REGION Network 56: Step[1130] : Gripper Forward
   RUNG wire#powerrail
      { S7_Templates := "SrcType := DInt" } EQ_Contact(in1 := "Unit1.Em7.ControlNodes".sepaGripper.sequence.status.currentStep, in2 := #JOB_11_STEP_30)
      Contact( "Unit1.Em7.ControlNodes".sepaGripper.sequence.status.seqActive )
      wire#w1
      Coil( "Unit1.Em7.ControlNodes".sepaGripper."step".action1[1130] )
   END_RUNG
   RUNG wire#w1
      Contact( "Unit1.Em7.ControlNodes".cmStackGripperFwdBwd.monitoring.inWorkPos )
      Coil( "Unit1.Em7.ControlNodes".sepaGripper."step".transition1[1130] )
   END_RUNG
   RUNG wire#w1
      Contact( "Unit1.Em7.ControlNodes".sepaGripper."step".transition1[1130] )
      Move(in := #JOB_11_STEP_40, out1 => "Unit1.Em7.ControlNodes".sepaGripper.sequence.status.nextStep)
   END_RUNG
   // the same network as SCL:
   "Unit1.Em7.ControlNodes".sepaGripper."step".action1[1130] := ("Unit1.Em7.ControlNodes".sepaGripper.sequence.status.currentStep = #JOB_11_STEP_30) AND "Unit1.Em7.ControlNodes".sepaGripper.sequence.status.seqActive;
   "Unit1.Em7.ControlNodes".sepaGripper."step".transition1[1130] := ("Unit1.Em7.ControlNodes".sepaGripper.sequence.status.currentStep = #JOB_11_STEP_30) AND "Unit1.Em7.ControlNodes".sepaGripper.sequence.status.seqActive AND "Unit1.Em7.ControlNodes".cmStackGripperFwdBwd.monitoring.inWorkPos;
   IF ("Unit1.Em7.ControlNodes".sepaGripper.sequence.status.currentStep = #JOB_11_STEP_30) AND "Unit1.Em7.ControlNodes".sepaGripper.sequence.status.seqActive AND "Unit1.Em7.ControlNodes".sepaGripper."step".transition1[1130] THEN
       "Unit1.Em7.ControlNodes".sepaGripper.sequence.status.nextStep := #JOB_11_STEP_40;
   END_IF;
END_REGION

REGION Network 57: Step[1140] : Gripper X-Axis Grip Pos
   RUNG wire#powerrail
      { S7_Templates := "SrcType := DInt" } EQ_Contact(in1 := "Unit1.Em7.ControlNodes".sepaGripper.sequence.status.currentStep, in2 := #JOB_11_STEP_40)
      Contact( "Unit1.Em7.ControlNodes".sepaGripper.sequence.status.seqActive )
      wire#w1
      Coil( "Unit1.Em7.ControlNodes".sepaGripper."step".action1[1140] )
   END_RUNG
   RUNG wire#w1
      Contact( "Unit1.Em7.ControlNodes".cm.softCam.sepaGripperAxisX.pickUpPOs.inPos )
      Coil( "Unit1.Em7.ControlNodes".sepaGripper."step".transition1[1140] )
   END_RUNG
   RUNG wire#w1
      Contact( "Unit1.Em7.ControlNodes".sepaGripper."step".transition1[1140] )
      Move(in := #JOB_11_STEP_90, out1 => "Unit1.Em7.ControlNodes".sepaGripper.sequence.status.nextStep)
   END_RUNG
   // the same network as SCL:
   "Unit1.Em7.ControlNodes".sepaGripper."step".action1[1140] := ("Unit1.Em7.ControlNodes".sepaGripper.sequence.status.currentStep = #JOB_11_STEP_40) AND "Unit1.Em7.ControlNodes".sepaGripper.sequence.status.seqActive;
   "Unit1.Em7.ControlNodes".sepaGripper."step".transition1[1140] := ("Unit1.Em7.ControlNodes".sepaGripper.sequence.status.currentStep = #JOB_11_STEP_40) AND "Unit1.Em7.ControlNodes".sepaGripper.sequence.status.seqActive AND "Unit1.Em7.ControlNodes".cm.softCam.sepaGripperAxisX.pickUpPOs.inPos;
   IF ("Unit1.Em7.ControlNodes".sepaGripper.sequence.status.currentStep = #JOB_11_STEP_40) AND "Unit1.Em7.ControlNodes".sepaGripper.sequence.status.seqActive AND "Unit1.Em7.ControlNodes".sepaGripper."step".transition1[1140] THEN
       "Unit1.Em7.ControlNodes".sepaGripper.sequence.status.nextStep := #JOB_11_STEP_90;
   END_IF;
END_REGION

REGION Network 58: Step[1190] : Job[11] Step End
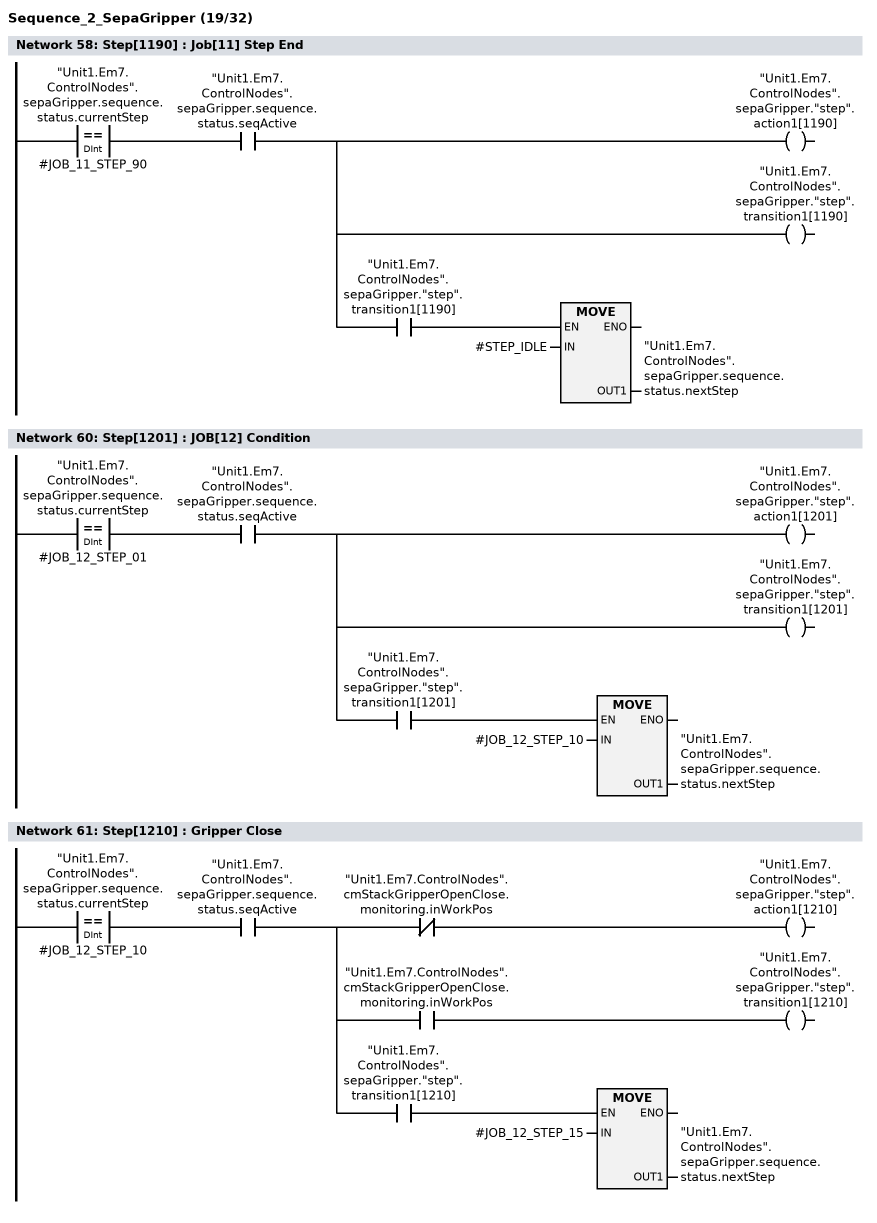
   RUNG wire#powerrail
      { S7_Templates := "SrcType := DInt" } EQ_Contact(in1 := "Unit1.Em7.ControlNodes".sepaGripper.sequence.status.currentStep, in2 := #JOB_11_STEP_90)
      Contact( "Unit1.Em7.ControlNodes".sepaGripper.sequence.status.seqActive )
      wire#w1
      Coil( "Unit1.Em7.ControlNodes".sepaGripper."step".action1[1190] )
   END_RUNG
   RUNG wire#w1
      Coil( "Unit1.Em7.ControlNodes".sepaGripper."step".transition1[1190] )
   END_RUNG
   RUNG wire#w1
      Contact( "Unit1.Em7.ControlNodes".sepaGripper."step".transition1[1190] )
      Move(in := #STEP_IDLE, out1 => "Unit1.Em7.ControlNodes".sepaGripper.sequence.status.nextStep)
   END_RUNG
   // the same network as SCL:
   "Unit1.Em7.ControlNodes".sepaGripper."step".action1[1190] := ("Unit1.Em7.ControlNodes".sepaGripper.sequence.status.currentStep = #JOB_11_STEP_90) AND "Unit1.Em7.ControlNodes".sepaGripper.sequence.status.seqActive;
   "Unit1.Em7.ControlNodes".sepaGripper."step".transition1[1190] := ("Unit1.Em7.ControlNodes".sepaGripper.sequence.status.currentStep = #JOB_11_STEP_90) AND "Unit1.Em7.ControlNodes".sepaGripper.sequence.status.seqActive;
   IF ("Unit1.Em7.ControlNodes".sepaGripper.sequence.status.currentStep = #JOB_11_STEP_90) AND "Unit1.Em7.ControlNodes".sepaGripper.sequence.status.seqActive AND "Unit1.Em7.ControlNodes".sepaGripper."step".transition1[1190] THEN
       "Unit1.Em7.ControlNodes".sepaGripper.sequence.status.nextStep := #STEP_IDLE;
   END_IF;
END_REGION

REGION Network 59: *************** JOB[12] Load To StackTable ************************
END_REGION

REGION Network 60: Step[1201] : JOB[12] Condition
   RUNG wire#powerrail
      { S7_Templates := "SrcType := DInt" } EQ_Contact(in1 := "Unit1.Em7.ControlNodes".sepaGripper.sequence.status.currentStep, in2 := #JOB_12_STEP_01)
      Contact( "Unit1.Em7.ControlNodes".sepaGripper.sequence.status.seqActive )
      wire#w1
      Coil( "Unit1.Em7.ControlNodes".sepaGripper."step".action1[1201] )
   END_RUNG
   RUNG wire#w1
      Coil( "Unit1.Em7.ControlNodes".sepaGripper."step".transition1[1201] )
   END_RUNG
   RUNG wire#w1
      Contact( "Unit1.Em7.ControlNodes".sepaGripper."step".transition1[1201] )
      Move(in := #JOB_12_STEP_10, out1 => "Unit1.Em7.ControlNodes".sepaGripper.sequence.status.nextStep)
   END_RUNG
   // the same network as SCL:
   "Unit1.Em7.ControlNodes".sepaGripper."step".action1[1201] := ("Unit1.Em7.ControlNodes".sepaGripper.sequence.status.currentStep = #JOB_12_STEP_01) AND "Unit1.Em7.ControlNodes".sepaGripper.sequence.status.seqActive;
   "Unit1.Em7.ControlNodes".sepaGripper."step".transition1[1201] := ("Unit1.Em7.ControlNodes".sepaGripper.sequence.status.currentStep = #JOB_12_STEP_01) AND "Unit1.Em7.ControlNodes".sepaGripper.sequence.status.seqActive;
   IF ("Unit1.Em7.ControlNodes".sepaGripper.sequence.status.currentStep = #JOB_12_STEP_01) AND "Unit1.Em7.ControlNodes".sepaGripper.sequence.status.seqActive AND "Unit1.Em7.ControlNodes".sepaGripper."step".transition1[1201] THEN
       "Unit1.Em7.ControlNodes".sepaGripper.sequence.status.nextStep := #JOB_12_STEP_10;
   END_IF;
END_REGION

REGION Network 61: Step[1210] : Gripper Close
   RUNG wire#powerrail
      { S7_Templates := "SrcType := DInt" } EQ_Contact(in1 := "Unit1.Em7.ControlNodes".sepaGripper.sequence.status.currentStep, in2 := #JOB_12_STEP_10)
      Contact( "Unit1.Em7.ControlNodes".sepaGripper.sequence.status.seqActive )
      wire#w1
      I_Contact( "Unit1.Em7.ControlNodes".cmStackGripperOpenClose.monitoring.inWorkPos )
      Coil( "Unit1.Em7.ControlNodes".sepaGripper."step".action1[1210] )
   END_RUNG
   RUNG wire#w1
      Contact( "Unit1.Em7.ControlNodes".cmStackGripperOpenClose.monitoring.inWorkPos )
      Coil( "Unit1.Em7.ControlNodes".sepaGripper."step".transition1[1210] )
   END_RUNG
   RUNG wire#w1
      Contact( "Unit1.Em7.ControlNodes".sepaGripper."step".transition1[1210] )
      Move(in := #JOB_12_STEP_15, out1 => "Unit1.Em7.ControlNodes".sepaGripper.sequence.status.nextStep)
   END_RUNG
   // the same network as SCL:
   #_w1 := ("Unit1.Em7.ControlNodes".sepaGripper.sequence.status.currentStep = #JOB_12_STEP_10) AND "Unit1.Em7.ControlNodes".sepaGripper.sequence.status.seqActive;
   "Unit1.Em7.ControlNodes".sepaGripper."step".action1[1210] := #_w1 AND NOT "Unit1.Em7.ControlNodes".cmStackGripperOpenClose.monitoring.inWorkPos;
   "Unit1.Em7.ControlNodes".sepaGripper."step".transition1[1210] := #_w1 AND "Unit1.Em7.ControlNodes".cmStackGripperOpenClose.monitoring.inWorkPos;
   IF #_w1 AND "Unit1.Em7.ControlNodes".sepaGripper."step".transition1[1210] THEN
       "Unit1.Em7.ControlNodes".sepaGripper.sequence.status.nextStep := #JOB_12_STEP_15;
   END_IF;
END_REGION

REGION Network 62: Step[1215] : Sepa Gripper → Stack Table [Loading Ready]
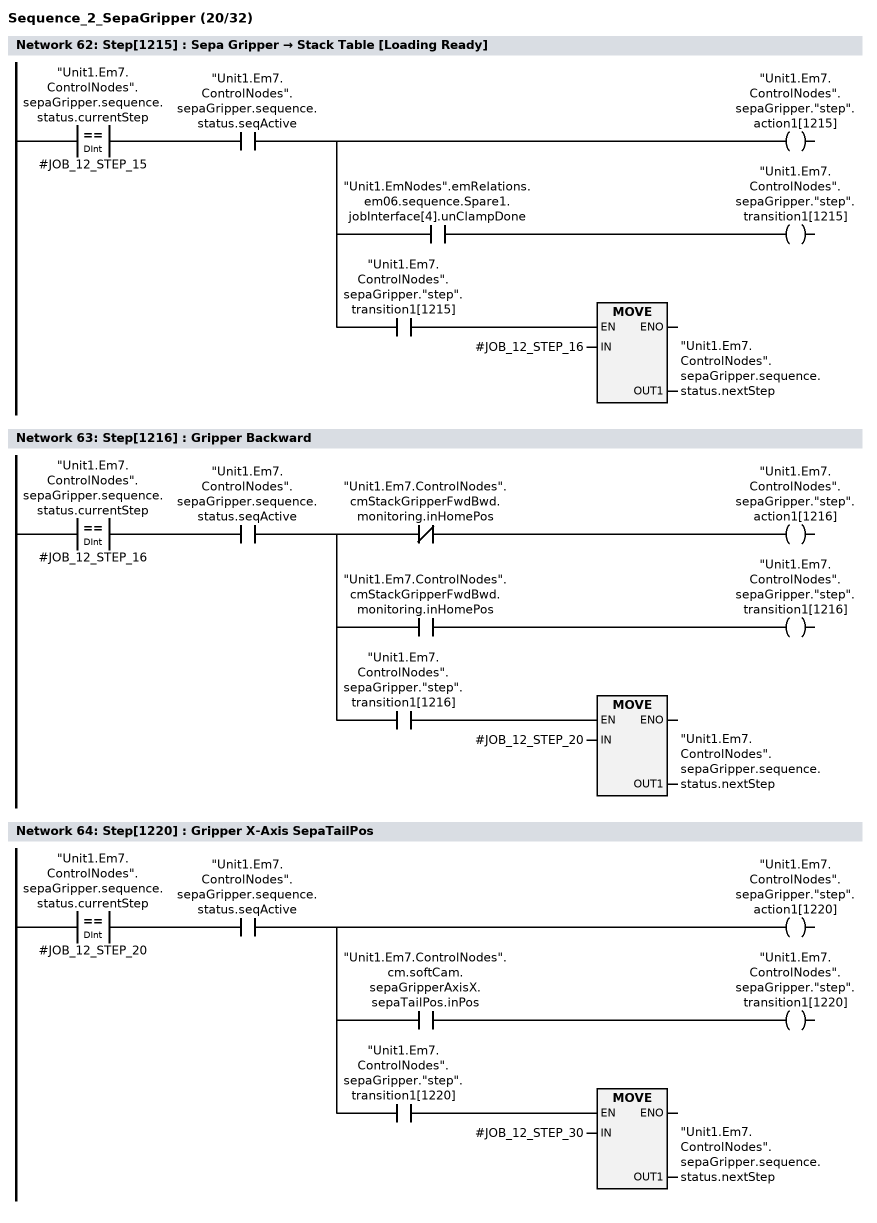
   RUNG wire#powerrail
      { S7_Templates := "SrcType := DInt" } EQ_Contact(in1 := "Unit1.Em7.ControlNodes".sepaGripper.sequence.status.currentStep, in2 := #JOB_12_STEP_15)
      Contact( "Unit1.Em7.ControlNodes".sepaGripper.sequence.status.seqActive )
      wire#w1
      Coil( "Unit1.Em7.ControlNodes".sepaGripper."step".action1[1215] )
   END_RUNG
   RUNG wire#w1
      Contact( "Unit1.EmNodes".emRelations.em06.sequence.Spare1.jobInterface[4].unClampDone )
      Coil( "Unit1.Em7.ControlNodes".sepaGripper."step".transition1[1215] )
   END_RUNG
   RUNG wire#w1
      Contact( "Unit1.Em7.ControlNodes".sepaGripper."step".transition1[1215] )
      Move(in := #JOB_12_STEP_16, out1 => "Unit1.Em7.ControlNodes".sepaGripper.sequence.status.nextStep)
   END_RUNG
   // the same network as SCL:
   "Unit1.Em7.ControlNodes".sepaGripper."step".action1[1215] := ("Unit1.Em7.ControlNodes".sepaGripper.sequence.status.currentStep = #JOB_12_STEP_15) AND "Unit1.Em7.ControlNodes".sepaGripper.sequence.status.seqActive;
   "Unit1.Em7.ControlNodes".sepaGripper."step".transition1[1215] := ("Unit1.Em7.ControlNodes".sepaGripper.sequence.status.currentStep = #JOB_12_STEP_15) AND "Unit1.Em7.ControlNodes".sepaGripper.sequence.status.seqActive AND "Unit1.EmNodes".emRelations.em06.sequence.Spare1.jobInterface[4].unClampDone;
   IF ("Unit1.Em7.ControlNodes".sepaGripper.sequence.status.currentStep = #JOB_12_STEP_15) AND "Unit1.Em7.ControlNodes".sepaGripper.sequence.status.seqActive AND "Unit1.Em7.ControlNodes".sepaGripper."step".transition1[1215] THEN
       "Unit1.Em7.ControlNodes".sepaGripper.sequence.status.nextStep := #JOB_12_STEP_16;
   END_IF;
END_REGION

REGION Network 63: Step[1216] : Gripper Backward
   RUNG wire#powerrail
      { S7_Templates := "SrcType := DInt" } EQ_Contact(in1 := "Unit1.Em7.ControlNodes".sepaGripper.sequence.status.currentStep, in2 := #JOB_12_STEP_16)
      Contact( "Unit1.Em7.ControlNodes".sepaGripper.sequence.status.seqActive )
      wire#w1
      I_Contact( "Unit1.Em7.ControlNodes".cmStackGripperFwdBwd.monitoring.inHomePos )
      Coil( "Unit1.Em7.ControlNodes".sepaGripper."step".action1[1216] )
   END_RUNG
   RUNG wire#w1
      Contact( "Unit1.Em7.ControlNodes".cmStackGripperFwdBwd.monitoring.inHomePos )
      Coil( "Unit1.Em7.ControlNodes".sepaGripper."step".transition1[1216] )
   END_RUNG
   RUNG wire#w1
      Contact( "Unit1.Em7.ControlNodes".sepaGripper."step".transition1[1216] )
      Move(in := #JOB_12_STEP_20, out1 => "Unit1.Em7.ControlNodes".sepaGripper.sequence.status.nextStep)
   END_RUNG
   // the same network as SCL:
   #_w1 := ("Unit1.Em7.ControlNodes".sepaGripper.sequence.status.currentStep = #JOB_12_STEP_16) AND "Unit1.Em7.ControlNodes".sepaGripper.sequence.status.seqActive;
   "Unit1.Em7.ControlNodes".sepaGripper."step".action1[1216] := #_w1 AND NOT "Unit1.Em7.ControlNodes".cmStackGripperFwdBwd.monitoring.inHomePos;
   "Unit1.Em7.ControlNodes".sepaGripper."step".transition1[1216] := #_w1 AND "Unit1.Em7.ControlNodes".cmStackGripperFwdBwd.monitoring.inHomePos;
   IF #_w1 AND "Unit1.Em7.ControlNodes".sepaGripper."step".transition1[1216] THEN
       "Unit1.Em7.ControlNodes".sepaGripper.sequence.status.nextStep := #JOB_12_STEP_20;
   END_IF;
END_REGION

REGION Network 64: Step[1220] : Gripper X-Axis SepaTailPos
   RUNG wire#powerrail
      { S7_Templates := "SrcType := DInt" } EQ_Contact(in1 := "Unit1.Em7.ControlNodes".sepaGripper.sequence.status.currentStep, in2 := #JOB_12_STEP_20)
      Contact( "Unit1.Em7.ControlNodes".sepaGripper.sequence.status.seqActive )
      wire#w1
      Coil( "Unit1.Em7.ControlNodes".sepaGripper."step".action1[1220] )
   END_RUNG
   RUNG wire#w1
      Contact( "Unit1.Em7.ControlNodes".cm.softCam.sepaGripperAxisX.sepaTailPos.inPos )
      Coil( "Unit1.Em7.ControlNodes".sepaGripper."step".transition1[1220] )
   END_RUNG
   RUNG wire#w1
      Contact( "Unit1.Em7.ControlNodes".sepaGripper."step".transition1[1220] )
      Move(in := #JOB_12_STEP_30, out1 => "Unit1.Em7.ControlNodes".sepaGripper.sequence.status.nextStep)
   END_RUNG
   // the same network as SCL:
   "Unit1.Em7.ControlNodes".sepaGripper."step".action1[1220] := ("Unit1.Em7.ControlNodes".sepaGripper.sequence.status.currentStep = #JOB_12_STEP_20) AND "Unit1.Em7.ControlNodes".sepaGripper.sequence.status.seqActive;
   "Unit1.Em7.ControlNodes".sepaGripper."step".transition1[1220] := ("Unit1.Em7.ControlNodes".sepaGripper.sequence.status.currentStep = #JOB_12_STEP_20) AND "Unit1.Em7.ControlNodes".sepaGripper.sequence.status.seqActive AND "Unit1.Em7.ControlNodes".cm.softCam.sepaGripperAxisX.sepaTailPos.inPos;
   IF ("Unit1.Em7.ControlNodes".sepaGripper.sequence.status.currentStep = #JOB_12_STEP_20) AND "Unit1.Em7.ControlNodes".sepaGripper.sequence.status.seqActive AND "Unit1.Em7.ControlNodes".sepaGripper."step".transition1[1220] THEN
       "Unit1.Em7.ControlNodes".sepaGripper.sequence.status.nextStep := #JOB_12_STEP_30;
   END_IF;
END_REGION

REGION Network 65: Step[1230] : Gripper Z-Axis Winder Pos
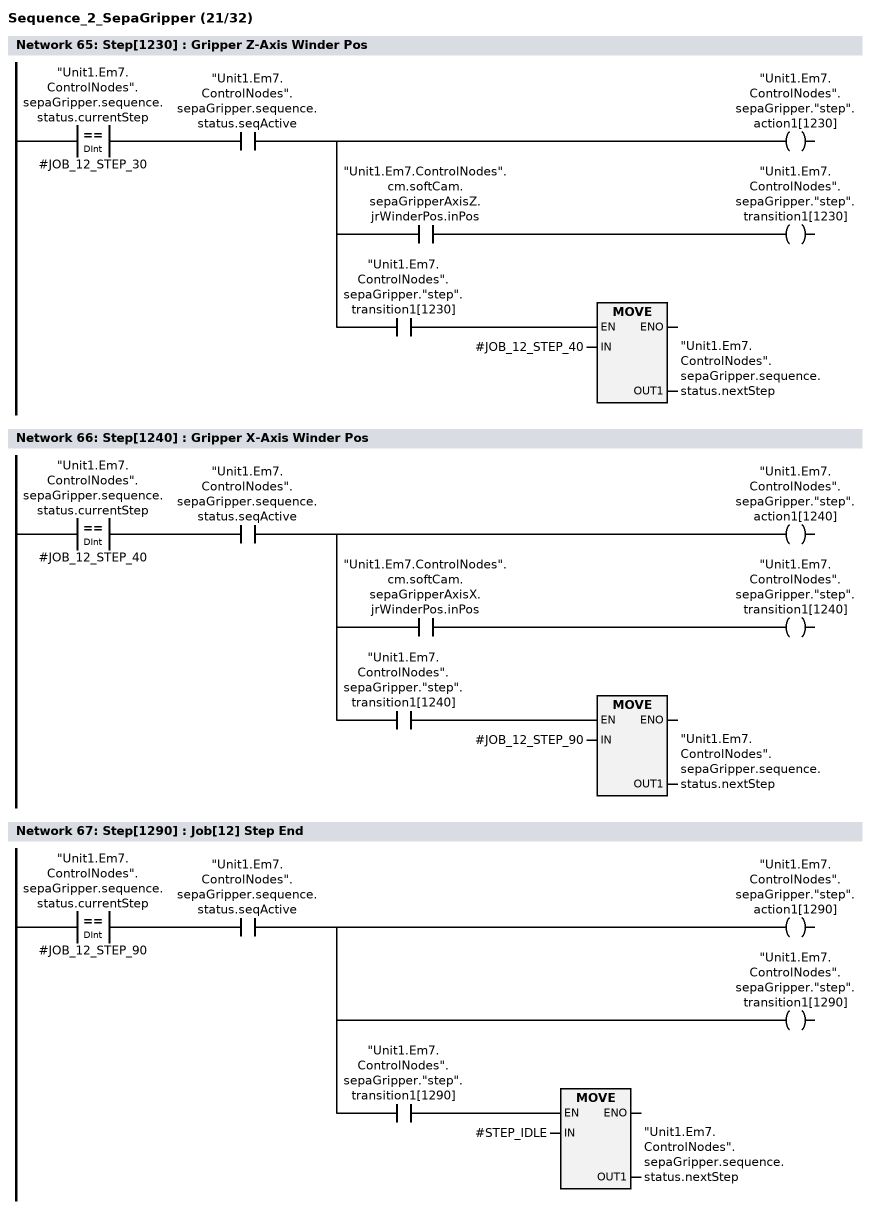
   RUNG wire#powerrail
      { S7_Templates := "SrcType := DInt" } EQ_Contact(in1 := "Unit1.Em7.ControlNodes".sepaGripper.sequence.status.currentStep, in2 := #JOB_12_STEP_30)
      Contact( "Unit1.Em7.ControlNodes".sepaGripper.sequence.status.seqActive )
      wire#w1
      Coil( "Unit1.Em7.ControlNodes".sepaGripper."step".action1[1230] )
   END_RUNG
   RUNG wire#w1
      Contact( "Unit1.Em7.ControlNodes".cm.softCam.sepaGripperAxisZ.jrWinderPos.inPos )
      Coil( "Unit1.Em7.ControlNodes".sepaGripper."step".transition1[1230] )
   END_RUNG
   RUNG wire#w1
      Contact( "Unit1.Em7.ControlNodes".sepaGripper."step".transition1[1230] )
      Move(in := #JOB_12_STEP_40, out1 => "Unit1.Em7.ControlNodes".sepaGripper.sequence.status.nextStep)
   END_RUNG
   // the same network as SCL:
   "Unit1.Em7.ControlNodes".sepaGripper."step".action1[1230] := ("Unit1.Em7.ControlNodes".sepaGripper.sequence.status.currentStep = #JOB_12_STEP_30) AND "Unit1.Em7.ControlNodes".sepaGripper.sequence.status.seqActive;
   "Unit1.Em7.ControlNodes".sepaGripper."step".transition1[1230] := ("Unit1.Em7.ControlNodes".sepaGripper.sequence.status.currentStep = #JOB_12_STEP_30) AND "Unit1.Em7.ControlNodes".sepaGripper.sequence.status.seqActive AND "Unit1.Em7.ControlNodes".cm.softCam.sepaGripperAxisZ.jrWinderPos.inPos;
   IF ("Unit1.Em7.ControlNodes".sepaGripper.sequence.status.currentStep = #JOB_12_STEP_30) AND "Unit1.Em7.ControlNodes".sepaGripper.sequence.status.seqActive AND "Unit1.Em7.ControlNodes".sepaGripper."step".transition1[1230] THEN
       "Unit1.Em7.ControlNodes".sepaGripper.sequence.status.nextStep := #JOB_12_STEP_40;
   END_IF;
END_REGION

REGION Network 66: Step[1240] : Gripper X-Axis Winder Pos
   RUNG wire#powerrail
      { S7_Templates := "SrcType := DInt" } EQ_Contact(in1 := "Unit1.Em7.ControlNodes".sepaGripper.sequence.status.currentStep, in2 := #JOB_12_STEP_40)
      Contact( "Unit1.Em7.ControlNodes".sepaGripper.sequence.status.seqActive )
      wire#w1
      Coil( "Unit1.Em7.ControlNodes".sepaGripper."step".action1[1240] )
   END_RUNG
   RUNG wire#w1
      Contact( "Unit1.Em7.ControlNodes".cm.softCam.sepaGripperAxisX.jrWinderPos.inPos )
      Coil( "Unit1.Em7.ControlNodes".sepaGripper."step".transition1[1240] )
   END_RUNG
   RUNG wire#w1
      Contact( "Unit1.Em7.ControlNodes".sepaGripper."step".transition1[1240] )
      Move(in := #JOB_12_STEP_90, out1 => "Unit1.Em7.ControlNodes".sepaGripper.sequence.status.nextStep)
   END_RUNG
   // the same network as SCL:
   "Unit1.Em7.ControlNodes".sepaGripper."step".action1[1240] := ("Unit1.Em7.ControlNodes".sepaGripper.sequence.status.currentStep = #JOB_12_STEP_40) AND "Unit1.Em7.ControlNodes".sepaGripper.sequence.status.seqActive;
   "Unit1.Em7.ControlNodes".sepaGripper."step".transition1[1240] := ("Unit1.Em7.ControlNodes".sepaGripper.sequence.status.currentStep = #JOB_12_STEP_40) AND "Unit1.Em7.ControlNodes".sepaGripper.sequence.status.seqActive AND "Unit1.Em7.ControlNodes".cm.softCam.sepaGripperAxisX.jrWinderPos.inPos;
   IF ("Unit1.Em7.ControlNodes".sepaGripper.sequence.status.currentStep = #JOB_12_STEP_40) AND "Unit1.Em7.ControlNodes".sepaGripper.sequence.status.seqActive AND "Unit1.Em7.ControlNodes".sepaGripper."step".transition1[1240] THEN
       "Unit1.Em7.ControlNodes".sepaGripper.sequence.status.nextStep := #JOB_12_STEP_90;
   END_IF;
END_REGION

REGION Network 67: Step[1290] : Job[12] Step End
   RUNG wire#powerrail
      { S7_Templates := "SrcType := DInt" } EQ_Contact(in1 := "Unit1.Em7.ControlNodes".sepaGripper.sequence.status.currentStep, in2 := #JOB_12_STEP_90)
      Contact( "Unit1.Em7.ControlNodes".sepaGripper.sequence.status.seqActive )
      wire#w1
      Coil( "Unit1.Em7.ControlNodes".sepaGripper."step".action1[1290] )
   END_RUNG
   RUNG wire#w1
      Coil( "Unit1.Em7.ControlNodes".sepaGripper."step".transition1[1290] )
   END_RUNG
   RUNG wire#w1
      Contact( "Unit1.Em7.ControlNodes".sepaGripper."step".transition1[1290] )
      Move(in := #STEP_IDLE, out1 => "Unit1.Em7.ControlNodes".sepaGripper.sequence.status.nextStep)
   END_RUNG
   // the same network as SCL:
   "Unit1.Em7.ControlNodes".sepaGripper."step".action1[1290] := ("Unit1.Em7.ControlNodes".sepaGripper.sequence.status.currentStep = #JOB_12_STEP_90) AND "Unit1.Em7.ControlNodes".sepaGripper.sequence.status.seqActive;
   "Unit1.Em7.ControlNodes".sepaGripper."step".transition1[1290] := ("Unit1.Em7.ControlNodes".sepaGripper.sequence.status.currentStep = #JOB_12_STEP_90) AND "Unit1.Em7.ControlNodes".sepaGripper.sequence.status.seqActive;
   IF ("Unit1.Em7.ControlNodes".sepaGripper.sequence.status.currentStep = #JOB_12_STEP_90) AND "Unit1.Em7.ControlNodes".sepaGripper.sequence.status.seqActive AND "Unit1.Em7.ControlNodes".sepaGripper."step".transition1[1290] THEN
       "Unit1.Em7.ControlNodes".sepaGripper.sequence.status.nextStep := #STEP_IDLE;
   END_IF;
END_REGION

REGION Network 68: *************** JOB[14] UnLoad To JRWinder ************************
END_REGION

REGION Network 69: Step[1401] : JOB[14] Condition
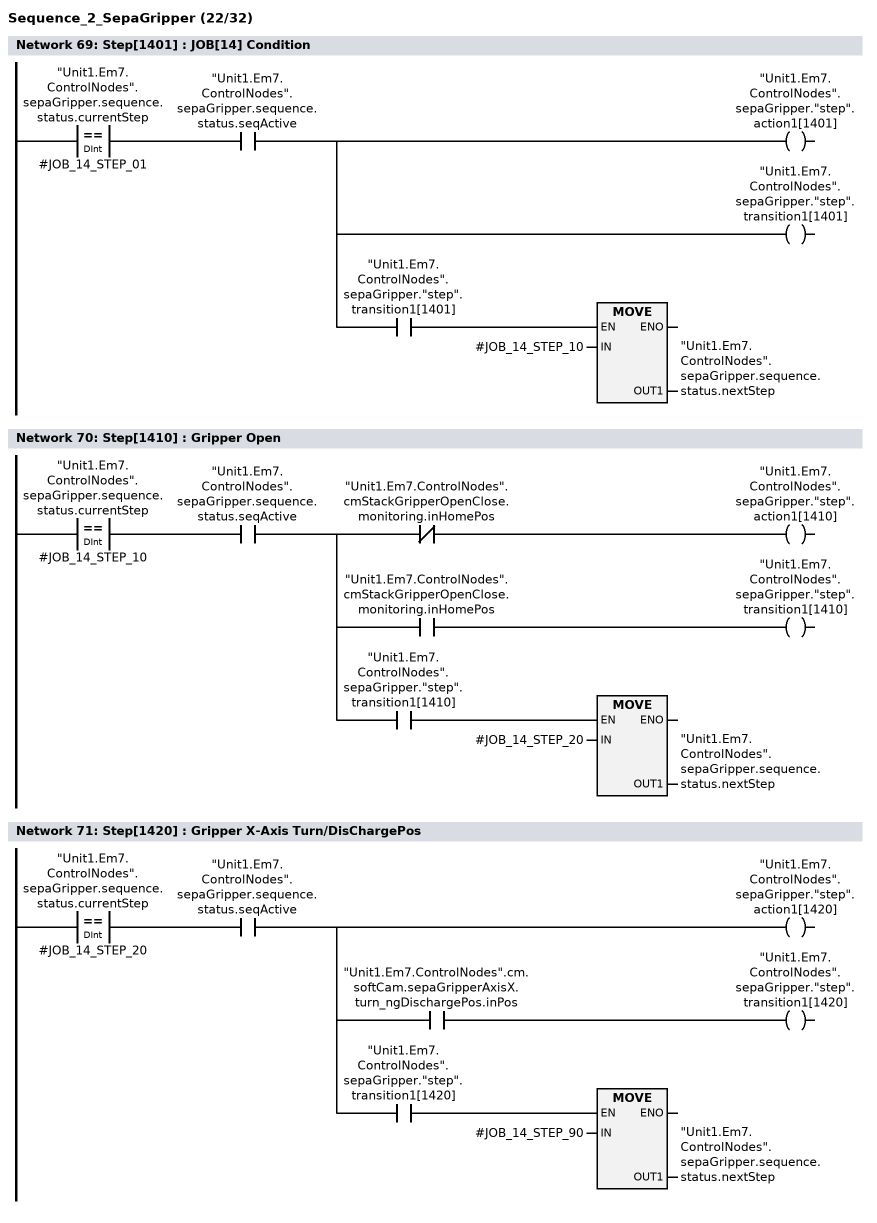
   RUNG wire#powerrail
      { S7_Templates := "SrcType := DInt" } EQ_Contact(in1 := "Unit1.Em7.ControlNodes".sepaGripper.sequence.status.currentStep, in2 := #JOB_14_STEP_01)
      Contact( "Unit1.Em7.ControlNodes".sepaGripper.sequence.status.seqActive )
      wire#w1
      Coil( "Unit1.Em7.ControlNodes".sepaGripper."step".action1[1401] )
   END_RUNG
   RUNG wire#w1
      Coil( "Unit1.Em7.ControlNodes".sepaGripper."step".transition1[1401] )
   END_RUNG
   RUNG wire#w1
      Contact( "Unit1.Em7.ControlNodes".sepaGripper."step".transition1[1401] )
      Move(in := #JOB_14_STEP_10, out1 => "Unit1.Em7.ControlNodes".sepaGripper.sequence.status.nextStep)
   END_RUNG
   // the same network as SCL:
   "Unit1.Em7.ControlNodes".sepaGripper."step".action1[1401] := ("Unit1.Em7.ControlNodes".sepaGripper.sequence.status.currentStep = #JOB_14_STEP_01) AND "Unit1.Em7.ControlNodes".sepaGripper.sequence.status.seqActive;
   "Unit1.Em7.ControlNodes".sepaGripper."step".transition1[1401] := ("Unit1.Em7.ControlNodes".sepaGripper.sequence.status.currentStep = #JOB_14_STEP_01) AND "Unit1.Em7.ControlNodes".sepaGripper.sequence.status.seqActive;
   IF ("Unit1.Em7.ControlNodes".sepaGripper.sequence.status.currentStep = #JOB_14_STEP_01) AND "Unit1.Em7.ControlNodes".sepaGripper.sequence.status.seqActive AND "Unit1.Em7.ControlNodes".sepaGripper."step".transition1[1401] THEN
       "Unit1.Em7.ControlNodes".sepaGripper.sequence.status.nextStep := #JOB_14_STEP_10;
   END_IF;
END_REGION

REGION Network 70: Step[1410] : Gripper Open
   RUNG wire#powerrail
      { S7_Templates := "SrcType := DInt" } EQ_Contact(in1 := "Unit1.Em7.ControlNodes".sepaGripper.sequence.status.currentStep, in2 := #JOB_14_STEP_10)
      Contact( "Unit1.Em7.ControlNodes".sepaGripper.sequence.status.seqActive )
      wire#w1
      I_Contact( "Unit1.Em7.ControlNodes".cmStackGripperOpenClose.monitoring.inHomePos )
      Coil( "Unit1.Em7.ControlNodes".sepaGripper."step".action1[1410] )
   END_RUNG
   RUNG wire#w1
      Contact( "Unit1.Em7.ControlNodes".cmStackGripperOpenClose.monitoring.inHomePos )
      Coil( "Unit1.Em7.ControlNodes".sepaGripper."step".transition1[1410] )
   END_RUNG
   RUNG wire#w1
      Contact( "Unit1.Em7.ControlNodes".sepaGripper."step".transition1[1410] )
      Move(in := #JOB_14_STEP_20, out1 => "Unit1.Em7.ControlNodes".sepaGripper.sequence.status.nextStep)
   END_RUNG
   // the same network as SCL:
   #_w1 := ("Unit1.Em7.ControlNodes".sepaGripper.sequence.status.currentStep = #JOB_14_STEP_10) AND "Unit1.Em7.ControlNodes".sepaGripper.sequence.status.seqActive;
   "Unit1.Em7.ControlNodes".sepaGripper."step".action1[1410] := #_w1 AND NOT "Unit1.Em7.ControlNodes".cmStackGripperOpenClose.monitoring.inHomePos;
   "Unit1.Em7.ControlNodes".sepaGripper."step".transition1[1410] := #_w1 AND "Unit1.Em7.ControlNodes".cmStackGripperOpenClose.monitoring.inHomePos;
   IF #_w1 AND "Unit1.Em7.ControlNodes".sepaGripper."step".transition1[1410] THEN
       "Unit1.Em7.ControlNodes".sepaGripper.sequence.status.nextStep := #JOB_14_STEP_20;
   END_IF;
END_REGION

REGION Network 71: Step[1420] : Gripper X-Axis Turn/DisChargePos
   RUNG wire#powerrail
      { S7_Templates := "SrcType := DInt" } EQ_Contact(in1 := "Unit1.Em7.ControlNodes".sepaGripper.sequence.status.currentStep, in2 := #JOB_14_STEP_20)
      Contact( "Unit1.Em7.ControlNodes".sepaGripper.sequence.status.seqActive )
      wire#w1
      Coil( "Unit1.Em7.ControlNodes".sepaGripper."step".action1[1420] )
   END_RUNG
   RUNG wire#w1
      Contact( "Unit1.Em7.ControlNodes".cm.softCam.sepaGripperAxisX.turn_ngDischargePos.inPos )
      Coil( "Unit1.Em7.ControlNodes".sepaGripper."step".transition1[1420] )
   END_RUNG
   RUNG wire#w1
      Contact( "Unit1.Em7.ControlNodes".sepaGripper."step".transition1[1420] )
      Move(in := #JOB_14_STEP_90, out1 => "Unit1.Em7.ControlNodes".sepaGripper.sequence.status.nextStep)
   END_RUNG
   // the same network as SCL:
   "Unit1.Em7.ControlNodes".sepaGripper."step".action1[1420] := ("Unit1.Em7.ControlNodes".sepaGripper.sequence.status.currentStep = #JOB_14_STEP_20) AND "Unit1.Em7.ControlNodes".sepaGripper.sequence.status.seqActive;
   "Unit1.Em7.ControlNodes".sepaGripper."step".transition1[1420] := ("Unit1.Em7.ControlNodes".sepaGripper.sequence.status.currentStep = #JOB_14_STEP_20) AND "Unit1.Em7.ControlNodes".sepaGripper.sequence.status.seqActive AND "Unit1.Em7.ControlNodes".cm.softCam.sepaGripperAxisX.turn_ngDischargePos.inPos;
   IF ("Unit1.Em7.ControlNodes".sepaGripper.sequence.status.currentStep = #JOB_14_STEP_20) AND "Unit1.Em7.ControlNodes".sepaGripper.sequence.status.seqActive AND "Unit1.Em7.ControlNodes".sepaGripper."step".transition1[1420] THEN
       "Unit1.Em7.ControlNodes".sepaGripper.sequence.status.nextStep := #JOB_14_STEP_90;
   END_IF;
END_REGION

REGION Network 72: Step[1490] : Job[14] Step End
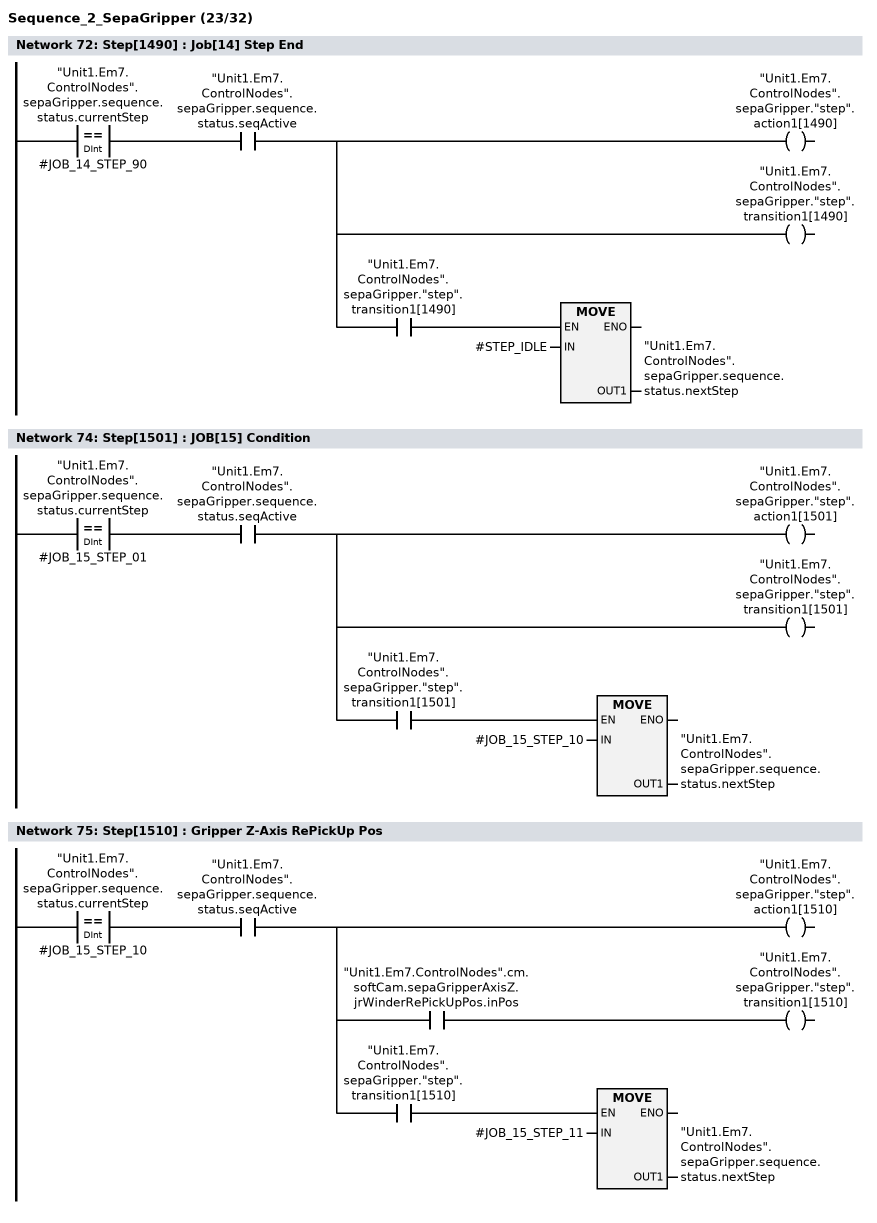
   RUNG wire#powerrail
      { S7_Templates := "SrcType := DInt" } EQ_Contact(in1 := "Unit1.Em7.ControlNodes".sepaGripper.sequence.status.currentStep, in2 := #JOB_14_STEP_90)
      Contact( "Unit1.Em7.ControlNodes".sepaGripper.sequence.status.seqActive )
      wire#w1
      Coil( "Unit1.Em7.ControlNodes".sepaGripper."step".action1[1490] )
   END_RUNG
   RUNG wire#w1
      Coil( "Unit1.Em7.ControlNodes".sepaGripper."step".transition1[1490] )
   END_RUNG
   RUNG wire#w1
      Contact( "Unit1.Em7.ControlNodes".sepaGripper."step".transition1[1490] )
      Move(in := #STEP_IDLE, out1 => "Unit1.Em7.ControlNodes".sepaGripper.sequence.status.nextStep)
   END_RUNG
   // the same network as SCL:
   "Unit1.Em7.ControlNodes".sepaGripper."step".action1[1490] := ("Unit1.Em7.ControlNodes".sepaGripper.sequence.status.currentStep = #JOB_14_STEP_90) AND "Unit1.Em7.ControlNodes".sepaGripper.sequence.status.seqActive;
   "Unit1.Em7.ControlNodes".sepaGripper."step".transition1[1490] := ("Unit1.Em7.ControlNodes".sepaGripper.sequence.status.currentStep = #JOB_14_STEP_90) AND "Unit1.Em7.ControlNodes".sepaGripper.sequence.status.seqActive;
   IF ("Unit1.Em7.ControlNodes".sepaGripper.sequence.status.currentStep = #JOB_14_STEP_90) AND "Unit1.Em7.ControlNodes".sepaGripper.sequence.status.seqActive AND "Unit1.Em7.ControlNodes".sepaGripper."step".transition1[1490] THEN
       "Unit1.Em7.ControlNodes".sepaGripper.sequence.status.nextStep := #STEP_IDLE;
   END_IF;
END_REGION

REGION Network 73: *************** JOB[15] Load To JRWinder ************************
END_REGION

REGION Network 74: Step[1501] : JOB[15] Condition
   RUNG wire#powerrail
      { S7_Templates := "SrcType := DInt" } EQ_Contact(in1 := "Unit1.Em7.ControlNodes".sepaGripper.sequence.status.currentStep, in2 := #JOB_15_STEP_01)
      Contact( "Unit1.Em7.ControlNodes".sepaGripper.sequence.status.seqActive )
      wire#w1
      Coil( "Unit1.Em7.ControlNodes".sepaGripper."step".action1[1501] )
   END_RUNG
   RUNG wire#w1
      Coil( "Unit1.Em7.ControlNodes".sepaGripper."step".transition1[1501] )
   END_RUNG
   RUNG wire#w1
      Contact( "Unit1.Em7.ControlNodes".sepaGripper."step".transition1[1501] )
      Move(in := #JOB_15_STEP_10, out1 => "Unit1.Em7.ControlNodes".sepaGripper.sequence.status.nextStep)
   END_RUNG
   // the same network as SCL:
   "Unit1.Em7.ControlNodes".sepaGripper."step".action1[1501] := ("Unit1.Em7.ControlNodes".sepaGripper.sequence.status.currentStep = #JOB_15_STEP_01) AND "Unit1.Em7.ControlNodes".sepaGripper.sequence.status.seqActive;
   "Unit1.Em7.ControlNodes".sepaGripper."step".transition1[1501] := ("Unit1.Em7.ControlNodes".sepaGripper.sequence.status.currentStep = #JOB_15_STEP_01) AND "Unit1.Em7.ControlNodes".sepaGripper.sequence.status.seqActive;
   IF ("Unit1.Em7.ControlNodes".sepaGripper.sequence.status.currentStep = #JOB_15_STEP_01) AND "Unit1.Em7.ControlNodes".sepaGripper.sequence.status.seqActive AND "Unit1.Em7.ControlNodes".sepaGripper."step".transition1[1501] THEN
       "Unit1.Em7.ControlNodes".sepaGripper.sequence.status.nextStep := #JOB_15_STEP_10;
   END_IF;
END_REGION

REGION Network 75: Step[1510] : Gripper Z-Axis RePickUp Pos
   RUNG wire#powerrail
      { S7_Templates := "SrcType := DInt" } EQ_Contact(in1 := "Unit1.Em7.ControlNodes".sepaGripper.sequence.status.currentStep, in2 := #JOB_15_STEP_10)
      Contact( "Unit1.Em7.ControlNodes".sepaGripper.sequence.status.seqActive )
      wire#w1
      Coil( "Unit1.Em7.ControlNodes".sepaGripper."step".action1[1510] )
   END_RUNG
   RUNG wire#w1
      Contact( "Unit1.Em7.ControlNodes".cm.softCam.sepaGripperAxisZ.jrWinderRePickUpPos.inPos )
      Coil( "Unit1.Em7.ControlNodes".sepaGripper."step".transition1[1510] )
   END_RUNG
   RUNG wire#w1
      Contact( "Unit1.Em7.ControlNodes".sepaGripper."step".transition1[1510] )
      Move(in := #JOB_15_STEP_11, out1 => "Unit1.Em7.ControlNodes".sepaGripper.sequence.status.nextStep)
   END_RUNG
   // the same network as SCL:
   "Unit1.Em7.ControlNodes".sepaGripper."step".action1[1510] := ("Unit1.Em7.ControlNodes".sepaGripper.sequence.status.currentStep = #JOB_15_STEP_10) AND "Unit1.Em7.ControlNodes".sepaGripper.sequence.status.seqActive;
   "Unit1.Em7.ControlNodes".sepaGripper."step".transition1[1510] := ("Unit1.Em7.ControlNodes".sepaGripper.sequence.status.currentStep = #JOB_15_STEP_10) AND "Unit1.Em7.ControlNodes".sepaGripper.sequence.status.seqActive AND "Unit1.Em7.ControlNodes".cm.softCam.sepaGripperAxisZ.jrWinderRePickUpPos.inPos;
   IF ("Unit1.Em7.ControlNodes".sepaGripper.sequence.status.currentStep = #JOB_15_STEP_10) AND "Unit1.Em7.ControlNodes".sepaGripper.sequence.status.seqActive AND "Unit1.Em7.ControlNodes".sepaGripper."step".transition1[1510] THEN
       "Unit1.Em7.ControlNodes".sepaGripper.sequence.status.nextStep := #JOB_15_STEP_11;
   END_IF;
END_REGION

REGION Network 76: Step[1511] : Gripper X-Axis Winder Pos
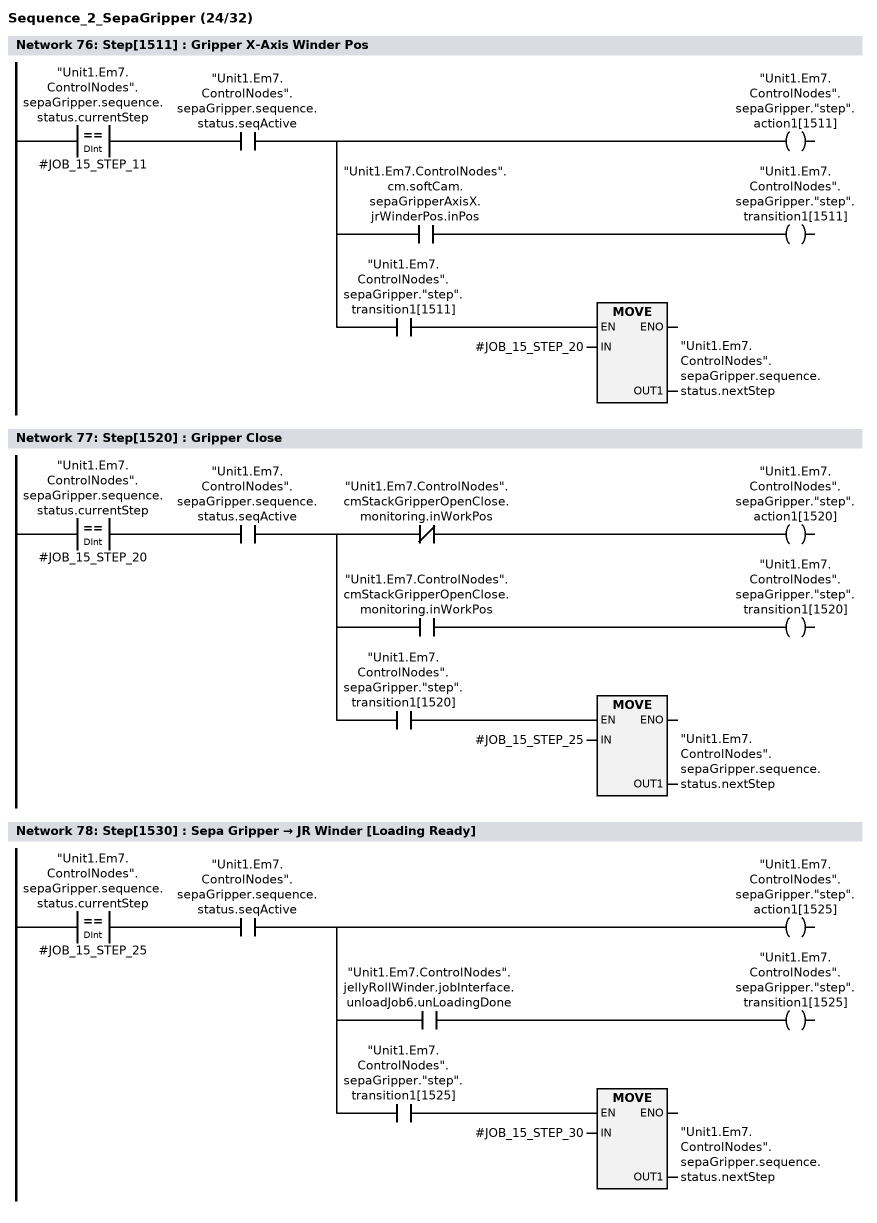
   RUNG wire#powerrail
      { S7_Templates := "SrcType := DInt" } EQ_Contact(in1 := "Unit1.Em7.ControlNodes".sepaGripper.sequence.status.currentStep, in2 := #JOB_15_STEP_11)
      Contact( "Unit1.Em7.ControlNodes".sepaGripper.sequence.status.seqActive )
      wire#w1
      Coil( "Unit1.Em7.ControlNodes".sepaGripper."step".action1[1511] )
   END_RUNG
   RUNG wire#w1
      Contact( "Unit1.Em7.ControlNodes".cm.softCam.sepaGripperAxisX.jrWinderPos.inPos )
      Coil( "Unit1.Em7.ControlNodes".sepaGripper."step".transition1[1511] )
   END_RUNG
   RUNG wire#w1
      Contact( "Unit1.Em7.ControlNodes".sepaGripper."step".transition1[1511] )
      Move(in := #JOB_15_STEP_20, out1 => "Unit1.Em7.ControlNodes".sepaGripper.sequence.status.nextStep)
   END_RUNG
   // the same network as SCL:
   "Unit1.Em7.ControlNodes".sepaGripper."step".action1[1511] := ("Unit1.Em7.ControlNodes".sepaGripper.sequence.status.currentStep = #JOB_15_STEP_11) AND "Unit1.Em7.ControlNodes".sepaGripper.sequence.status.seqActive;
   "Unit1.Em7.ControlNodes".sepaGripper."step".transition1[1511] := ("Unit1.Em7.ControlNodes".sepaGripper.sequence.status.currentStep = #JOB_15_STEP_11) AND "Unit1.Em7.ControlNodes".sepaGripper.sequence.status.seqActive AND "Unit1.Em7.ControlNodes".cm.softCam.sepaGripperAxisX.jrWinderPos.inPos;
   IF ("Unit1.Em7.ControlNodes".sepaGripper.sequence.status.currentStep = #JOB_15_STEP_11) AND "Unit1.Em7.ControlNodes".sepaGripper.sequence.status.seqActive AND "Unit1.Em7.ControlNodes".sepaGripper."step".transition1[1511] THEN
       "Unit1.Em7.ControlNodes".sepaGripper.sequence.status.nextStep := #JOB_15_STEP_20;
   END_IF;
END_REGION

REGION Network 77: Step[1520] : Gripper Close
   RUNG wire#powerrail
      { S7_Templates := "SrcType := DInt" } EQ_Contact(in1 := "Unit1.Em7.ControlNodes".sepaGripper.sequence.status.currentStep, in2 := #JOB_15_STEP_20)
      Contact( "Unit1.Em7.ControlNodes".sepaGripper.sequence.status.seqActive )
      wire#w1
      I_Contact( "Unit1.Em7.ControlNodes".cmStackGripperOpenClose.monitoring.inWorkPos )
      Coil( "Unit1.Em7.ControlNodes".sepaGripper."step".action1[1520] )
   END_RUNG
   RUNG wire#w1
      Contact( "Unit1.Em7.ControlNodes".cmStackGripperOpenClose.monitoring.inWorkPos )
      Coil( "Unit1.Em7.ControlNodes".sepaGripper."step".transition1[1520] )
   END_RUNG
   RUNG wire#w1
      Contact( "Unit1.Em7.ControlNodes".sepaGripper."step".transition1[1520] )
      Move(in := #JOB_15_STEP_25, out1 => "Unit1.Em7.ControlNodes".sepaGripper.sequence.status.nextStep)
   END_RUNG
   // the same network as SCL:
   #_w1 := ("Unit1.Em7.ControlNodes".sepaGripper.sequence.status.currentStep = #JOB_15_STEP_20) AND "Unit1.Em7.ControlNodes".sepaGripper.sequence.status.seqActive;
   "Unit1.Em7.ControlNodes".sepaGripper."step".action1[1520] := #_w1 AND NOT "Unit1.Em7.ControlNodes".cmStackGripperOpenClose.monitoring.inWorkPos;
   "Unit1.Em7.ControlNodes".sepaGripper."step".transition1[1520] := #_w1 AND "Unit1.Em7.ControlNodes".cmStackGripperOpenClose.monitoring.inWorkPos;
   IF #_w1 AND "Unit1.Em7.ControlNodes".sepaGripper."step".transition1[1520] THEN
       "Unit1.Em7.ControlNodes".sepaGripper.sequence.status.nextStep := #JOB_15_STEP_25;
   END_IF;
END_REGION

REGION Network 78: Step[1530] : Sepa Gripper → JR Winder [Loading Ready]
   RUNG wire#powerrail
      { S7_Templates := "SrcType := DInt" } EQ_Contact(in1 := "Unit1.Em7.ControlNodes".sepaGripper.sequence.status.currentStep, in2 := #JOB_15_STEP_25)
      Contact( "Unit1.Em7.ControlNodes".sepaGripper.sequence.status.seqActive )
      wire#w1
      Coil( "Unit1.Em7.ControlNodes".sepaGripper."step".action1[1525] )
   END_RUNG
   RUNG wire#w1
      Contact( "Unit1.Em7.ControlNodes".jellyRollWinder.jobInterface.unloadJob6.unLoadingDone )
      Coil( "Unit1.Em7.ControlNodes".sepaGripper."step".transition1[1525] )
   END_RUNG
   RUNG wire#w1
      Contact( "Unit1.Em7.ControlNodes".sepaGripper."step".transition1[1525] )
      Move(in := #JOB_15_STEP_30, out1 => "Unit1.Em7.ControlNodes".sepaGripper.sequence.status.nextStep)
   END_RUNG
   // the same network as SCL:
   "Unit1.Em7.ControlNodes".sepaGripper."step".action1[1525] := ("Unit1.Em7.ControlNodes".sepaGripper.sequence.status.currentStep = #JOB_15_STEP_25) AND "Unit1.Em7.ControlNodes".sepaGripper.sequence.status.seqActive;
   "Unit1.Em7.ControlNodes".sepaGripper."step".transition1[1525] := ("Unit1.Em7.ControlNodes".sepaGripper.sequence.status.currentStep = #JOB_15_STEP_25) AND "Unit1.Em7.ControlNodes".sepaGripper.sequence.status.seqActive AND "Unit1.Em7.ControlNodes".jellyRollWinder.jobInterface.unloadJob6.unLoadingDone;
   IF ("Unit1.Em7.ControlNodes".sepaGripper.sequence.status.currentStep = #JOB_15_STEP_25) AND "Unit1.Em7.ControlNodes".sepaGripper.sequence.status.seqActive AND "Unit1.Em7.ControlNodes".sepaGripper."step".transition1[1525] THEN
       "Unit1.Em7.ControlNodes".sepaGripper.sequence.status.nextStep := #JOB_15_STEP_30;
   END_IF;
END_REGION

REGION Network 79: Step[1530] : Gripper X-Axis Turn/Discharge Pos
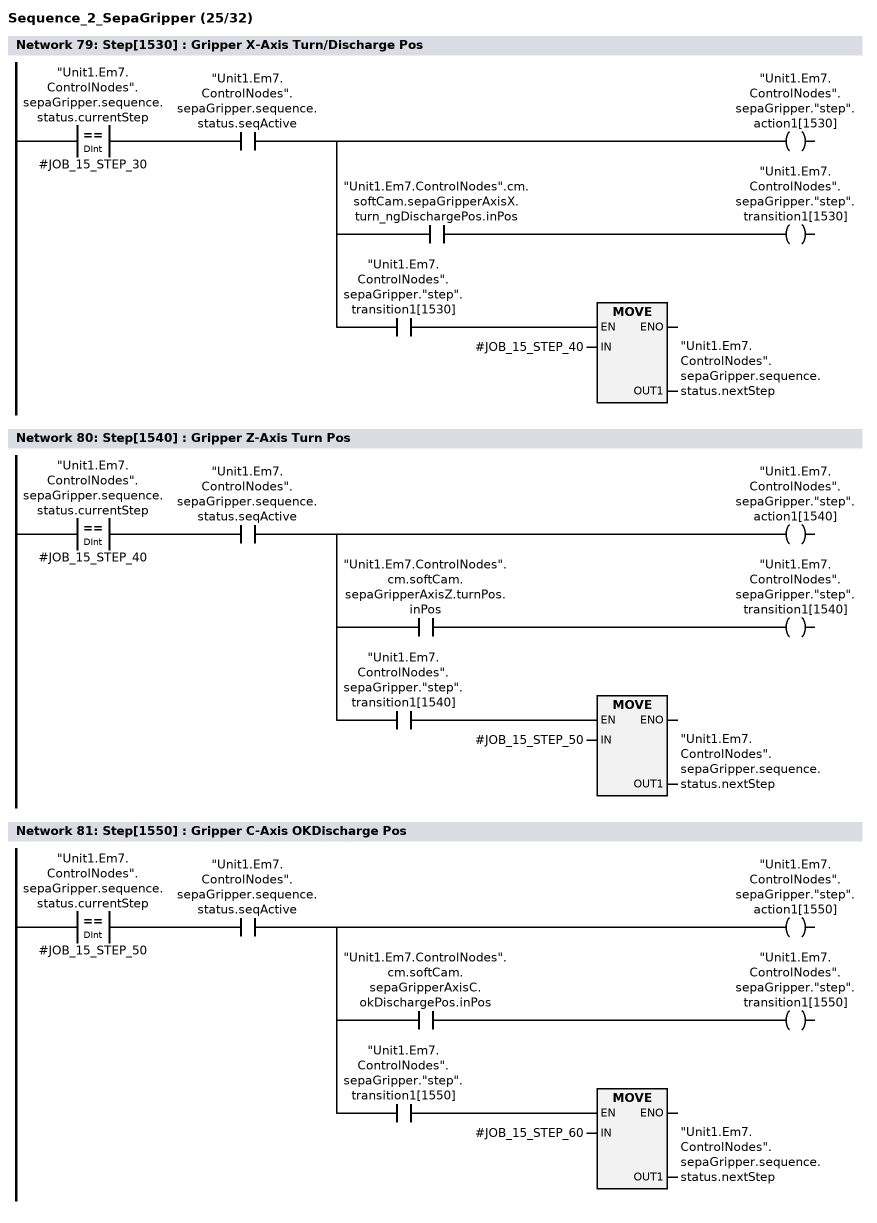
   RUNG wire#powerrail
      { S7_Templates := "SrcType := DInt" } EQ_Contact(in1 := "Unit1.Em7.ControlNodes".sepaGripper.sequence.status.currentStep, in2 := #JOB_15_STEP_30)
      Contact( "Unit1.Em7.ControlNodes".sepaGripper.sequence.status.seqActive )
      wire#w1
      Coil( "Unit1.Em7.ControlNodes".sepaGripper."step".action1[1530] )
   END_RUNG
   RUNG wire#w1
      Contact( "Unit1.Em7.ControlNodes".cm.softCam.sepaGripperAxisX.turn_ngDischargePos.inPos )
      Coil( "Unit1.Em7.ControlNodes".sepaGripper."step".transition1[1530] )
   END_RUNG
   RUNG wire#w1
      Contact( "Unit1.Em7.ControlNodes".sepaGripper."step".transition1[1530] )
      Move(in := #JOB_15_STEP_40, out1 => "Unit1.Em7.ControlNodes".sepaGripper.sequence.status.nextStep)
   END_RUNG
   // the same network as SCL:
   "Unit1.Em7.ControlNodes".sepaGripper."step".action1[1530] := ("Unit1.Em7.ControlNodes".sepaGripper.sequence.status.currentStep = #JOB_15_STEP_30) AND "Unit1.Em7.ControlNodes".sepaGripper.sequence.status.seqActive;
   "Unit1.Em7.ControlNodes".sepaGripper."step".transition1[1530] := ("Unit1.Em7.ControlNodes".sepaGripper.sequence.status.currentStep = #JOB_15_STEP_30) AND "Unit1.Em7.ControlNodes".sepaGripper.sequence.status.seqActive AND "Unit1.Em7.ControlNodes".cm.softCam.sepaGripperAxisX.turn_ngDischargePos.inPos;
   IF ("Unit1.Em7.ControlNodes".sepaGripper.sequence.status.currentStep = #JOB_15_STEP_30) AND "Unit1.Em7.ControlNodes".sepaGripper.sequence.status.seqActive AND "Unit1.Em7.ControlNodes".sepaGripper."step".transition1[1530] THEN
       "Unit1.Em7.ControlNodes".sepaGripper.sequence.status.nextStep := #JOB_15_STEP_40;
   END_IF;
END_REGION

REGION Network 80: Step[1540] : Gripper Z-Axis Turn Pos
   RUNG wire#powerrail
      { S7_Templates := "SrcType := DInt" } EQ_Contact(in1 := "Unit1.Em7.ControlNodes".sepaGripper.sequence.status.currentStep, in2 := #JOB_15_STEP_40)
      Contact( "Unit1.Em7.ControlNodes".sepaGripper.sequence.status.seqActive )
      wire#w1
      Coil( "Unit1.Em7.ControlNodes".sepaGripper."step".action1[1540] )
   END_RUNG
   RUNG wire#w1
      Contact( "Unit1.Em7.ControlNodes".cm.softCam.sepaGripperAxisZ.turnPos.inPos )
      Coil( "Unit1.Em7.ControlNodes".sepaGripper."step".transition1[1540] )
   END_RUNG
   RUNG wire#w1
      Contact( "Unit1.Em7.ControlNodes".sepaGripper."step".transition1[1540] )
      Move(in := #JOB_15_STEP_50, out1 => "Unit1.Em7.ControlNodes".sepaGripper.sequence.status.nextStep)
   END_RUNG
   // the same network as SCL:
   "Unit1.Em7.ControlNodes".sepaGripper."step".action1[1540] := ("Unit1.Em7.ControlNodes".sepaGripper.sequence.status.currentStep = #JOB_15_STEP_40) AND "Unit1.Em7.ControlNodes".sepaGripper.sequence.status.seqActive;
   "Unit1.Em7.ControlNodes".sepaGripper."step".transition1[1540] := ("Unit1.Em7.ControlNodes".sepaGripper.sequence.status.currentStep = #JOB_15_STEP_40) AND "Unit1.Em7.ControlNodes".sepaGripper.sequence.status.seqActive AND "Unit1.Em7.ControlNodes".cm.softCam.sepaGripperAxisZ.turnPos.inPos;
   IF ("Unit1.Em7.ControlNodes".sepaGripper.sequence.status.currentStep = #JOB_15_STEP_40) AND "Unit1.Em7.ControlNodes".sepaGripper.sequence.status.seqActive AND "Unit1.Em7.ControlNodes".sepaGripper."step".transition1[1540] THEN
       "Unit1.Em7.ControlNodes".sepaGripper.sequence.status.nextStep := #JOB_15_STEP_50;
   END_IF;
END_REGION

REGION Network 81: Step[1550] : Gripper C-Axis OKDischarge Pos
   RUNG wire#powerrail
      { S7_Templates := "SrcType := DInt" } EQ_Contact(in1 := "Unit1.Em7.ControlNodes".sepaGripper.sequence.status.currentStep, in2 := #JOB_15_STEP_50)
      Contact( "Unit1.Em7.ControlNodes".sepaGripper.sequence.status.seqActive )
      wire#w1
      Coil( "Unit1.Em7.ControlNodes".sepaGripper."step".action1[1550] )
   END_RUNG
   RUNG wire#w1
      Contact( "Unit1.Em7.ControlNodes".cm.softCam.sepaGripperAxisC.okDischargePos.inPos )
      Coil( "Unit1.Em7.ControlNodes".sepaGripper."step".transition1[1550] )
   END_RUNG
   RUNG wire#w1
      Contact( "Unit1.Em7.ControlNodes".sepaGripper."step".transition1[1550] )
      Move(in := #JOB_15_STEP_60, out1 => "Unit1.Em7.ControlNodes".sepaGripper.sequence.status.nextStep)
   END_RUNG
   // the same network as SCL:
   "Unit1.Em7.ControlNodes".sepaGripper."step".action1[1550] := ("Unit1.Em7.ControlNodes".sepaGripper.sequence.status.currentStep = #JOB_15_STEP_50) AND "Unit1.Em7.ControlNodes".sepaGripper.sequence.status.seqActive;
   "Unit1.Em7.ControlNodes".sepaGripper."step".transition1[1550] := ("Unit1.Em7.ControlNodes".sepaGripper.sequence.status.currentStep = #JOB_15_STEP_50) AND "Unit1.Em7.ControlNodes".sepaGripper.sequence.status.seqActive AND "Unit1.Em7.ControlNodes".cm.softCam.sepaGripperAxisC.okDischargePos.inPos;
   IF ("Unit1.Em7.ControlNodes".sepaGripper.sequence.status.currentStep = #JOB_15_STEP_50) AND "Unit1.Em7.ControlNodes".sepaGripper.sequence.status.seqActive AND "Unit1.Em7.ControlNodes".sepaGripper."step".transition1[1550] THEN
       "Unit1.Em7.ControlNodes".sepaGripper.sequence.status.nextStep := #JOB_15_STEP_60;
   END_IF;
END_REGION

REGION Network 82: Step[1560] : Gripper Z-Axis OKDischarge Pos
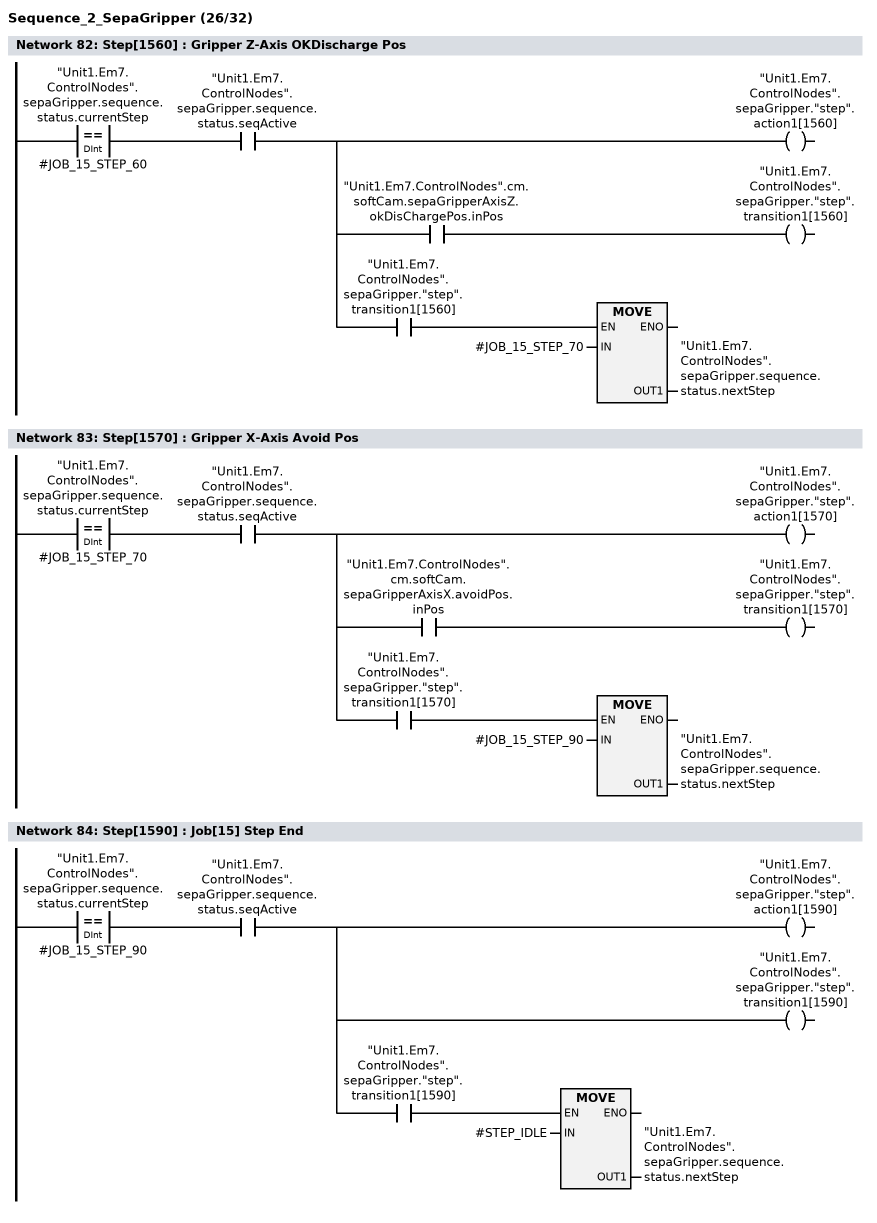
   RUNG wire#powerrail
      { S7_Templates := "SrcType := DInt" } EQ_Contact(in1 := "Unit1.Em7.ControlNodes".sepaGripper.sequence.status.currentStep, in2 := #JOB_15_STEP_60)
      Contact( "Unit1.Em7.ControlNodes".sepaGripper.sequence.status.seqActive )
      wire#w1
      Coil( "Unit1.Em7.ControlNodes".sepaGripper."step".action1[1560] )
   END_RUNG
   RUNG wire#w1
      Contact( "Unit1.Em7.ControlNodes".cm.softCam.sepaGripperAxisZ.okDisChargePos.inPos )
      Coil( "Unit1.Em7.ControlNodes".sepaGripper."step".transition1[1560] )
   END_RUNG
   RUNG wire#w1
      Contact( "Unit1.Em7.ControlNodes".sepaGripper."step".transition1[1560] )
      Move(in := #JOB_15_STEP_70, out1 => "Unit1.Em7.ControlNodes".sepaGripper.sequence.status.nextStep)
   END_RUNG
   // the same network as SCL:
   "Unit1.Em7.ControlNodes".sepaGripper."step".action1[1560] := ("Unit1.Em7.ControlNodes".sepaGripper.sequence.status.currentStep = #JOB_15_STEP_60) AND "Unit1.Em7.ControlNodes".sepaGripper.sequence.status.seqActive;
   "Unit1.Em7.ControlNodes".sepaGripper."step".transition1[1560] := ("Unit1.Em7.ControlNodes".sepaGripper.sequence.status.currentStep = #JOB_15_STEP_60) AND "Unit1.Em7.ControlNodes".sepaGripper.sequence.status.seqActive AND "Unit1.Em7.ControlNodes".cm.softCam.sepaGripperAxisZ.okDisChargePos.inPos;
   IF ("Unit1.Em7.ControlNodes".sepaGripper.sequence.status.currentStep = #JOB_15_STEP_60) AND "Unit1.Em7.ControlNodes".sepaGripper.sequence.status.seqActive AND "Unit1.Em7.ControlNodes".sepaGripper."step".transition1[1560] THEN
       "Unit1.Em7.ControlNodes".sepaGripper.sequence.status.nextStep := #JOB_15_STEP_70;
   END_IF;
END_REGION

REGION Network 83: Step[1570] : Gripper X-Axis Avoid Pos
   RUNG wire#powerrail
      { S7_Templates := "SrcType := DInt" } EQ_Contact(in1 := "Unit1.Em7.ControlNodes".sepaGripper.sequence.status.currentStep, in2 := #JOB_15_STEP_70)
      Contact( "Unit1.Em7.ControlNodes".sepaGripper.sequence.status.seqActive )
      wire#w1
      Coil( "Unit1.Em7.ControlNodes".sepaGripper."step".action1[1570] )
   END_RUNG
   RUNG wire#w1
      Contact( "Unit1.Em7.ControlNodes".cm.softCam.sepaGripperAxisX.avoidPos.inPos )
      Coil( "Unit1.Em7.ControlNodes".sepaGripper."step".transition1[1570] )
   END_RUNG
   RUNG wire#w1
      Contact( "Unit1.Em7.ControlNodes".sepaGripper."step".transition1[1570] )
      Move(in := #JOB_15_STEP_90, out1 => "Unit1.Em7.ControlNodes".sepaGripper.sequence.status.nextStep)
   END_RUNG
   // the same network as SCL:
   "Unit1.Em7.ControlNodes".sepaGripper."step".action1[1570] := ("Unit1.Em7.ControlNodes".sepaGripper.sequence.status.currentStep = #JOB_15_STEP_70) AND "Unit1.Em7.ControlNodes".sepaGripper.sequence.status.seqActive;
   "Unit1.Em7.ControlNodes".sepaGripper."step".transition1[1570] := ("Unit1.Em7.ControlNodes".sepaGripper.sequence.status.currentStep = #JOB_15_STEP_70) AND "Unit1.Em7.ControlNodes".sepaGripper.sequence.status.seqActive AND "Unit1.Em7.ControlNodes".cm.softCam.sepaGripperAxisX.avoidPos.inPos;
   IF ("Unit1.Em7.ControlNodes".sepaGripper.sequence.status.currentStep = #JOB_15_STEP_70) AND "Unit1.Em7.ControlNodes".sepaGripper.sequence.status.seqActive AND "Unit1.Em7.ControlNodes".sepaGripper."step".transition1[1570] THEN
       "Unit1.Em7.ControlNodes".sepaGripper.sequence.status.nextStep := #JOB_15_STEP_90;
   END_IF;
END_REGION

REGION Network 84: Step[1590] : Job[15] Step End
   RUNG wire#powerrail
      { S7_Templates := "SrcType := DInt" } EQ_Contact(in1 := "Unit1.Em7.ControlNodes".sepaGripper.sequence.status.currentStep, in2 := #JOB_15_STEP_90)
      Contact( "Unit1.Em7.ControlNodes".sepaGripper.sequence.status.seqActive )
      wire#w1
      Coil( "Unit1.Em7.ControlNodes".sepaGripper."step".action1[1590] )
   END_RUNG
   RUNG wire#w1
      Coil( "Unit1.Em7.ControlNodes".sepaGripper."step".transition1[1590] )
   END_RUNG
   RUNG wire#w1
      Contact( "Unit1.Em7.ControlNodes".sepaGripper."step".transition1[1590] )
      Move(in := #STEP_IDLE, out1 => "Unit1.Em7.ControlNodes".sepaGripper.sequence.status.nextStep)
   END_RUNG
   // the same network as SCL:
   "Unit1.Em7.ControlNodes".sepaGripper."step".action1[1590] := ("Unit1.Em7.ControlNodes".sepaGripper.sequence.status.currentStep = #JOB_15_STEP_90) AND "Unit1.Em7.ControlNodes".sepaGripper.sequence.status.seqActive;
   "Unit1.Em7.ControlNodes".sepaGripper."step".transition1[1590] := ("Unit1.Em7.ControlNodes".sepaGripper.sequence.status.currentStep = #JOB_15_STEP_90) AND "Unit1.Em7.ControlNodes".sepaGripper.sequence.status.seqActive;
   IF ("Unit1.Em7.ControlNodes".sepaGripper.sequence.status.currentStep = #JOB_15_STEP_90) AND "Unit1.Em7.ControlNodes".sepaGripper.sequence.status.seqActive AND "Unit1.Em7.ControlNodes".sepaGripper."step".transition1[1590] THEN
       "Unit1.Em7.ControlNodes".sepaGripper.sequence.status.nextStep := #STEP_IDLE;
   END_IF;
END_REGION

REGION Network 85: *************** JOB[17] Unload To Inspection ************************
END_REGION

REGION Network 86: Step[1701] : JOB[17] Condition
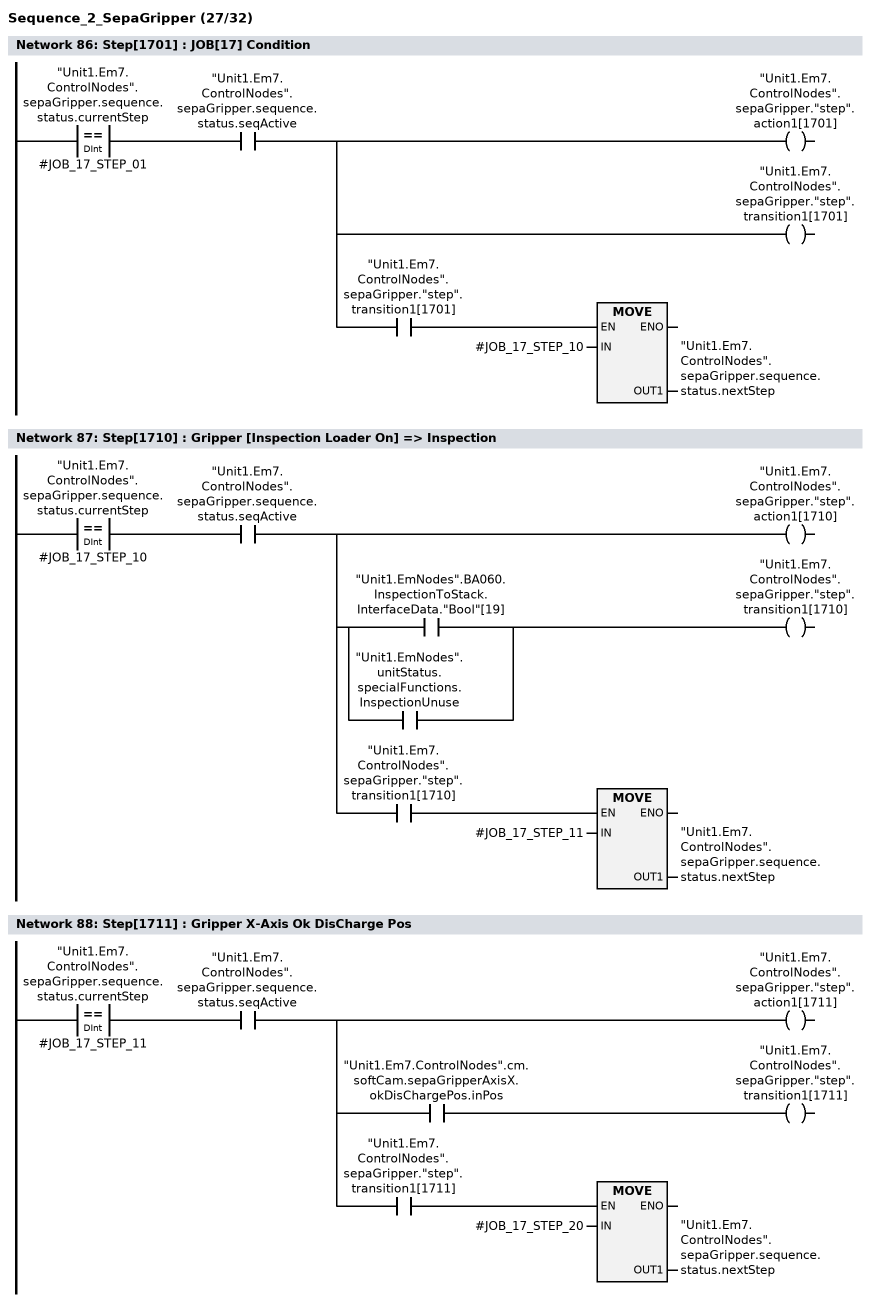
   RUNG wire#powerrail
      { S7_Templates := "SrcType := DInt" } EQ_Contact(in1 := "Unit1.Em7.ControlNodes".sepaGripper.sequence.status.currentStep, in2 := #JOB_17_STEP_01)
      Contact( "Unit1.Em7.ControlNodes".sepaGripper.sequence.status.seqActive )
      wire#w1
      Coil( "Unit1.Em7.ControlNodes".sepaGripper."step".action1[1701] )
   END_RUNG
   RUNG wire#w1
      Coil( "Unit1.Em7.ControlNodes".sepaGripper."step".transition1[1701] )
   END_RUNG
   RUNG wire#w1
      Contact( "Unit1.Em7.ControlNodes".sepaGripper."step".transition1[1701] )
      Move(in := #JOB_17_STEP_10, out1 => "Unit1.Em7.ControlNodes".sepaGripper.sequence.status.nextStep)
   END_RUNG
   // the same network as SCL:
   "Unit1.Em7.ControlNodes".sepaGripper."step".action1[1701] := ("Unit1.Em7.ControlNodes".sepaGripper.sequence.status.currentStep = #JOB_17_STEP_01) AND "Unit1.Em7.ControlNodes".sepaGripper.sequence.status.seqActive;
   "Unit1.Em7.ControlNodes".sepaGripper."step".transition1[1701] := ("Unit1.Em7.ControlNodes".sepaGripper.sequence.status.currentStep = #JOB_17_STEP_01) AND "Unit1.Em7.ControlNodes".sepaGripper.sequence.status.seqActive;
   IF ("Unit1.Em7.ControlNodes".sepaGripper.sequence.status.currentStep = #JOB_17_STEP_01) AND "Unit1.Em7.ControlNodes".sepaGripper.sequence.status.seqActive AND "Unit1.Em7.ControlNodes".sepaGripper."step".transition1[1701] THEN
       "Unit1.Em7.ControlNodes".sepaGripper.sequence.status.nextStep := #JOB_17_STEP_10;
   END_IF;
END_REGION

REGION Network 87: Step[1710] : Gripper [Inspection Loader On] => Inspection
   RUNG wire#powerrail
      { S7_Templates := "SrcType := DInt" } EQ_Contact(in1 := "Unit1.Em7.ControlNodes".sepaGripper.sequence.status.currentStep, in2 := #JOB_17_STEP_10)
      Contact( "Unit1.Em7.ControlNodes".sepaGripper.sequence.status.seqActive )
      wire#w1
      Coil( "Unit1.Em7.ControlNodes".sepaGripper."step".action1[1710] )
   END_RUNG
   RUNG wire#w1
      Contact( "Unit1.EmNodes".BA060.InspectionToStack.InterfaceData."Bool"[19] )
      wire#w2
      Coil( "Unit1.Em7.ControlNodes".sepaGripper."step".transition1[1710] )
   END_RUNG
   RUNG wire#w1
      Contact( "Unit1.EmNodes".unitStatus.specialFunctions.InspectionUnuse )
   END_RUNG wire#w2
   RUNG wire#w1
      Contact( "Unit1.Em7.ControlNodes".sepaGripper."step".transition1[1710] )
      Move(in := #JOB_17_STEP_11, out1 => "Unit1.Em7.ControlNodes".sepaGripper.sequence.status.nextStep)
   END_RUNG
   // the same network as SCL:
   "Unit1.Em7.ControlNodes".sepaGripper."step".action1[1710] := ("Unit1.Em7.ControlNodes".sepaGripper.sequence.status.currentStep = #JOB_17_STEP_10) AND "Unit1.Em7.ControlNodes".sepaGripper.sequence.status.seqActive;
   "Unit1.Em7.ControlNodes".sepaGripper."step".transition1[1710] := ("Unit1.Em7.ControlNodes".sepaGripper.sequence.status.currentStep = #JOB_17_STEP_10) AND "Unit1.Em7.ControlNodes".sepaGripper.sequence.status.seqActive AND ("Unit1.EmNodes".BA060.InspectionToStack.InterfaceData."Bool"[19] OR "Unit1.EmNodes".unitStatus.specialFunctions.InspectionUnuse);
   IF ("Unit1.Em7.ControlNodes".sepaGripper.sequence.status.currentStep = #JOB_17_STEP_10) AND "Unit1.Em7.ControlNodes".sepaGripper.sequence.status.seqActive AND "Unit1.Em7.ControlNodes".sepaGripper."step".transition1[1710] THEN
       "Unit1.Em7.ControlNodes".sepaGripper.sequence.status.nextStep := #JOB_17_STEP_11;
   END_IF;
END_REGION

REGION Network 88: Step[1711] : Gripper X-Axis Ok DisCharge Pos
   RUNG wire#powerrail
      { S7_Templates := "SrcType := DInt" } EQ_Contact(in1 := "Unit1.Em7.ControlNodes".sepaGripper.sequence.status.currentStep, in2 := #JOB_17_STEP_11)
      Contact( "Unit1.Em7.ControlNodes".sepaGripper.sequence.status.seqActive )
      wire#w1
      Coil( "Unit1.Em7.ControlNodes".sepaGripper."step".action1[1711] )
   END_RUNG
   RUNG wire#w1
      Contact( "Unit1.Em7.ControlNodes".cm.softCam.sepaGripperAxisX.okDisChargePos.inPos )
      Coil( "Unit1.Em7.ControlNodes".sepaGripper."step".transition1[1711] )
   END_RUNG
   RUNG wire#w1
      Contact( "Unit1.Em7.ControlNodes".sepaGripper."step".transition1[1711] )
      Move(in := #JOB_17_STEP_20, out1 => "Unit1.Em7.ControlNodes".sepaGripper.sequence.status.nextStep)
   END_RUNG
   // the same network as SCL:
   "Unit1.Em7.ControlNodes".sepaGripper."step".action1[1711] := ("Unit1.Em7.ControlNodes".sepaGripper.sequence.status.currentStep = #JOB_17_STEP_11) AND "Unit1.Em7.ControlNodes".sepaGripper.sequence.status.seqActive;
   "Unit1.Em7.ControlNodes".sepaGripper."step".transition1[1711] := ("Unit1.Em7.ControlNodes".sepaGripper.sequence.status.currentStep = #JOB_17_STEP_11) AND "Unit1.Em7.ControlNodes".sepaGripper.sequence.status.seqActive AND "Unit1.Em7.ControlNodes".cm.softCam.sepaGripperAxisX.okDisChargePos.inPos;
   IF ("Unit1.Em7.ControlNodes".sepaGripper.sequence.status.currentStep = #JOB_17_STEP_11) AND "Unit1.Em7.ControlNodes".sepaGripper.sequence.status.seqActive AND "Unit1.Em7.ControlNodes".sepaGripper."step".transition1[1711] THEN
       "Unit1.Em7.ControlNodes".sepaGripper.sequence.status.nextStep := #JOB_17_STEP_20;
   END_IF;
END_REGION

REGION Network 89: Step[1720] : Gripper [Inspection UnClamp Req] => Inspection
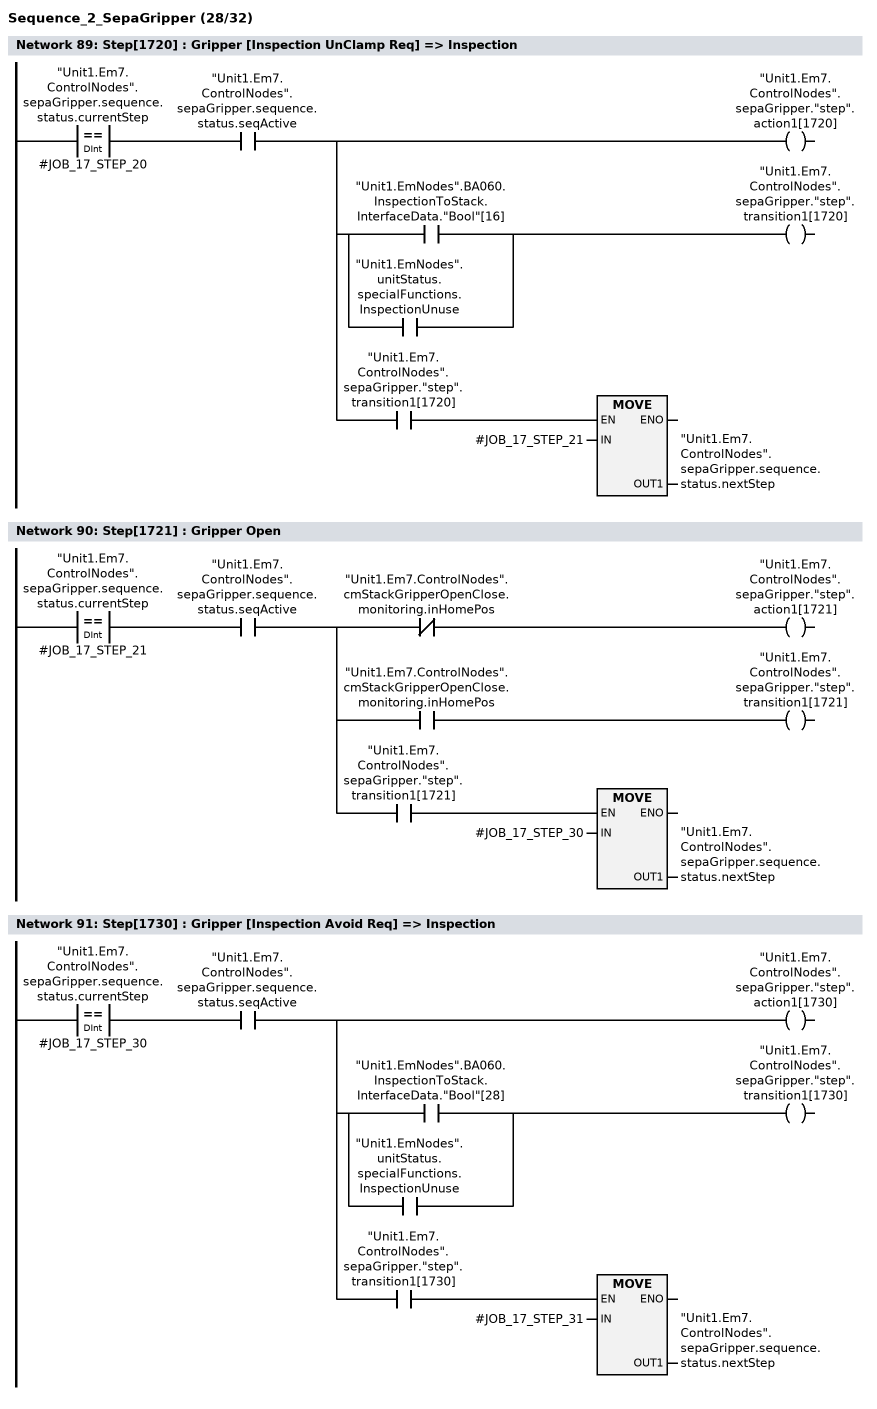
   RUNG wire#powerrail
      { S7_Templates := "SrcType := DInt" } EQ_Contact(in1 := "Unit1.Em7.ControlNodes".sepaGripper.sequence.status.currentStep, in2 := #JOB_17_STEP_20)
      Contact( "Unit1.Em7.ControlNodes".sepaGripper.sequence.status.seqActive )
      wire#w1
      Coil( "Unit1.Em7.ControlNodes".sepaGripper."step".action1[1720] )
   END_RUNG
   RUNG wire#w1
      Contact( "Unit1.EmNodes".BA060.InspectionToStack.InterfaceData."Bool"[16] )
      wire#w2
      Coil( "Unit1.Em7.ControlNodes".sepaGripper."step".transition1[1720] )
   END_RUNG
   RUNG wire#w1
      Contact( "Unit1.EmNodes".unitStatus.specialFunctions.InspectionUnuse )
   END_RUNG wire#w2
   RUNG wire#w1
      Contact( "Unit1.Em7.ControlNodes".sepaGripper."step".transition1[1720] )
      Move(in := #JOB_17_STEP_21, out1 => "Unit1.Em7.ControlNodes".sepaGripper.sequence.status.nextStep)
   END_RUNG
   // the same network as SCL:
   "Unit1.Em7.ControlNodes".sepaGripper."step".action1[1720] := ("Unit1.Em7.ControlNodes".sepaGripper.sequence.status.currentStep = #JOB_17_STEP_20) AND "Unit1.Em7.ControlNodes".sepaGripper.sequence.status.seqActive;
   "Unit1.Em7.ControlNodes".sepaGripper."step".transition1[1720] := ("Unit1.Em7.ControlNodes".sepaGripper.sequence.status.currentStep = #JOB_17_STEP_20) AND "Unit1.Em7.ControlNodes".sepaGripper.sequence.status.seqActive AND ("Unit1.EmNodes".BA060.InspectionToStack.InterfaceData."Bool"[16] OR "Unit1.EmNodes".unitStatus.specialFunctions.InspectionUnuse);
   IF ("Unit1.Em7.ControlNodes".sepaGripper.sequence.status.currentStep = #JOB_17_STEP_20) AND "Unit1.Em7.ControlNodes".sepaGripper.sequence.status.seqActive AND "Unit1.Em7.ControlNodes".sepaGripper."step".transition1[1720] THEN
       "Unit1.Em7.ControlNodes".sepaGripper.sequence.status.nextStep := #JOB_17_STEP_21;
   END_IF;
END_REGION

REGION Network 90: Step[1721] : Gripper Open
   RUNG wire#powerrail
      { S7_Templates := "SrcType := DInt" } EQ_Contact(in1 := "Unit1.Em7.ControlNodes".sepaGripper.sequence.status.currentStep, in2 := #JOB_17_STEP_21)
      Contact( "Unit1.Em7.ControlNodes".sepaGripper.sequence.status.seqActive )
      wire#w1
      I_Contact( "Unit1.Em7.ControlNodes".cmStackGripperOpenClose.monitoring.inHomePos )
      Coil( "Unit1.Em7.ControlNodes".sepaGripper."step".action1[1721] )
   END_RUNG
   RUNG wire#w1
      Contact( "Unit1.Em7.ControlNodes".cmStackGripperOpenClose.monitoring.inHomePos )
      Coil( "Unit1.Em7.ControlNodes".sepaGripper."step".transition1[1721] )
   END_RUNG
   RUNG wire#w1
      Contact( "Unit1.Em7.ControlNodes".sepaGripper."step".transition1[1721] )
      Move(in := #JOB_17_STEP_30, out1 => "Unit1.Em7.ControlNodes".sepaGripper.sequence.status.nextStep)
   END_RUNG
   // the same network as SCL:
   #_w1 := ("Unit1.Em7.ControlNodes".sepaGripper.sequence.status.currentStep = #JOB_17_STEP_21) AND "Unit1.Em7.ControlNodes".sepaGripper.sequence.status.seqActive;
   "Unit1.Em7.ControlNodes".sepaGripper."step".action1[1721] := #_w1 AND NOT "Unit1.Em7.ControlNodes".cmStackGripperOpenClose.monitoring.inHomePos;
   "Unit1.Em7.ControlNodes".sepaGripper."step".transition1[1721] := #_w1 AND "Unit1.Em7.ControlNodes".cmStackGripperOpenClose.monitoring.inHomePos;
   IF #_w1 AND "Unit1.Em7.ControlNodes".sepaGripper."step".transition1[1721] THEN
       "Unit1.Em7.ControlNodes".sepaGripper.sequence.status.nextStep := #JOB_17_STEP_30;
   END_IF;
END_REGION

REGION Network 91: Step[1730] : Gripper [Inspection Avoid Req] => Inspection
   RUNG wire#powerrail
      { S7_Templates := "SrcType := DInt" } EQ_Contact(in1 := "Unit1.Em7.ControlNodes".sepaGripper.sequence.status.currentStep, in2 := #JOB_17_STEP_30)
      Contact( "Unit1.Em7.ControlNodes".sepaGripper.sequence.status.seqActive )
      wire#w1
      Coil( "Unit1.Em7.ControlNodes".sepaGripper."step".action1[1730] )
   END_RUNG
   RUNG wire#w1
      Contact( "Unit1.EmNodes".BA060.InspectionToStack.InterfaceData."Bool"[28] )
      wire#w2
      Coil( "Unit1.Em7.ControlNodes".sepaGripper."step".transition1[1730] )
   END_RUNG
   RUNG wire#w1
      Contact( "Unit1.EmNodes".unitStatus.specialFunctions.InspectionUnuse )
   END_RUNG wire#w2
   RUNG wire#w1
      Contact( "Unit1.Em7.ControlNodes".sepaGripper."step".transition1[1730] )
      Move(in := #JOB_17_STEP_31, out1 => "Unit1.Em7.ControlNodes".sepaGripper.sequence.status.nextStep)
   END_RUNG
   // the same network as SCL:
   "Unit1.Em7.ControlNodes".sepaGripper."step".action1[1730] := ("Unit1.Em7.ControlNodes".sepaGripper.sequence.status.currentStep = #JOB_17_STEP_30) AND "Unit1.Em7.ControlNodes".sepaGripper.sequence.status.seqActive;
   "Unit1.Em7.ControlNodes".sepaGripper."step".transition1[1730] := ("Unit1.Em7.ControlNodes".sepaGripper.sequence.status.currentStep = #JOB_17_STEP_30) AND "Unit1.Em7.ControlNodes".sepaGripper.sequence.status.seqActive AND ("Unit1.EmNodes".BA060.InspectionToStack.InterfaceData."Bool"[28] OR "Unit1.EmNodes".unitStatus.specialFunctions.InspectionUnuse);
   IF ("Unit1.Em7.ControlNodes".sepaGripper.sequence.status.currentStep = #JOB_17_STEP_30) AND "Unit1.Em7.ControlNodes".sepaGripper.sequence.status.seqActive AND "Unit1.Em7.ControlNodes".sepaGripper."step".transition1[1730] THEN
       "Unit1.Em7.ControlNodes".sepaGripper.sequence.status.nextStep := #JOB_17_STEP_31;
   END_IF;
END_REGION

REGION Network 92: Step[1731] : Gripper X-Axis Avoid Pos
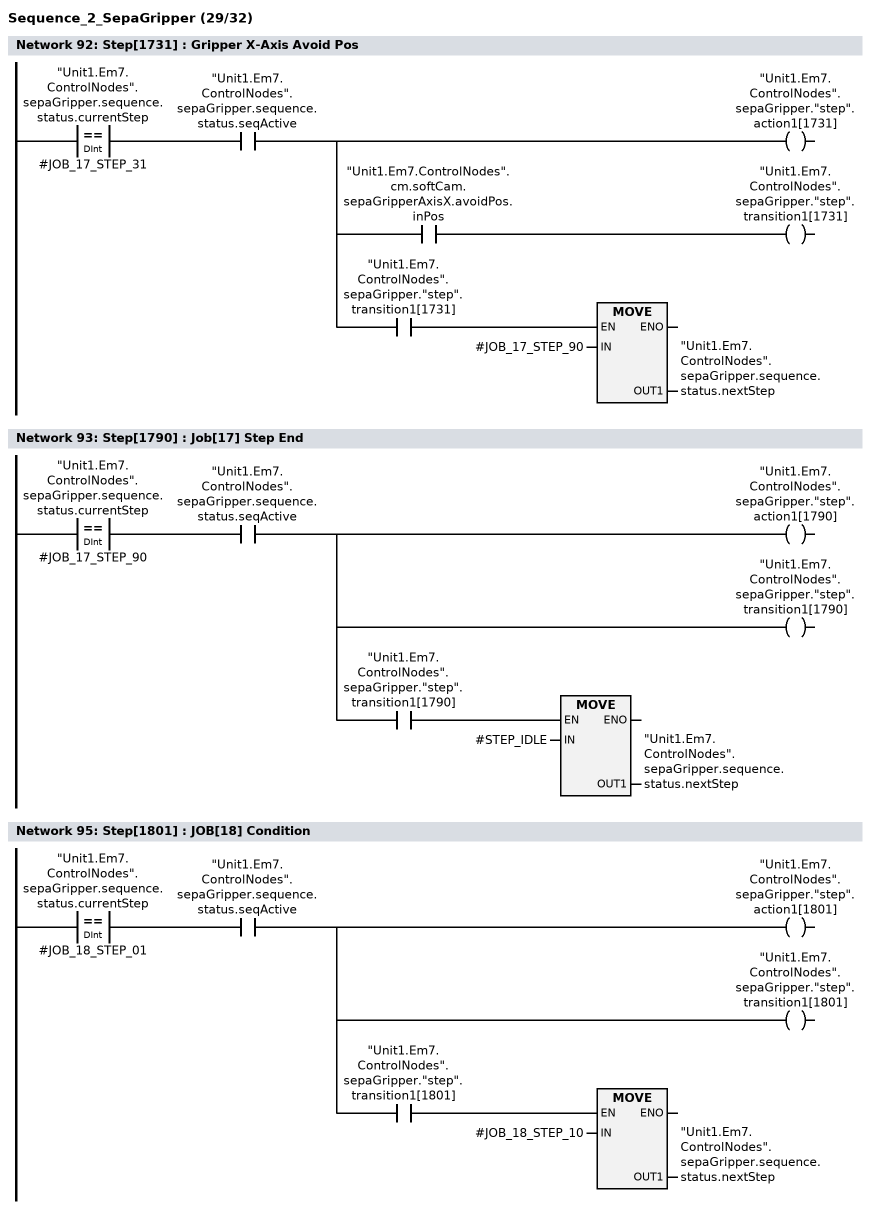
   RUNG wire#powerrail
      { S7_Templates := "SrcType := DInt" } EQ_Contact(in1 := "Unit1.Em7.ControlNodes".sepaGripper.sequence.status.currentStep, in2 := #JOB_17_STEP_31)
      Contact( "Unit1.Em7.ControlNodes".sepaGripper.sequence.status.seqActive )
      wire#w1
      Coil( "Unit1.Em7.ControlNodes".sepaGripper."step".action1[1731] )
   END_RUNG
   RUNG wire#w1
      Contact( "Unit1.Em7.ControlNodes".cm.softCam.sepaGripperAxisX.avoidPos.inPos )
      Coil( "Unit1.Em7.ControlNodes".sepaGripper."step".transition1[1731] )
   END_RUNG
   RUNG wire#w1
      Contact( "Unit1.Em7.ControlNodes".sepaGripper."step".transition1[1731] )
      Move(in := #JOB_17_STEP_90, out1 => "Unit1.Em7.ControlNodes".sepaGripper.sequence.status.nextStep)
   END_RUNG
   // the same network as SCL:
   "Unit1.Em7.ControlNodes".sepaGripper."step".action1[1731] := ("Unit1.Em7.ControlNodes".sepaGripper.sequence.status.currentStep = #JOB_17_STEP_31) AND "Unit1.Em7.ControlNodes".sepaGripper.sequence.status.seqActive;
   "Unit1.Em7.ControlNodes".sepaGripper."step".transition1[1731] := ("Unit1.Em7.ControlNodes".sepaGripper.sequence.status.currentStep = #JOB_17_STEP_31) AND "Unit1.Em7.ControlNodes".sepaGripper.sequence.status.seqActive AND "Unit1.Em7.ControlNodes".cm.softCam.sepaGripperAxisX.avoidPos.inPos;
   IF ("Unit1.Em7.ControlNodes".sepaGripper.sequence.status.currentStep = #JOB_17_STEP_31) AND "Unit1.Em7.ControlNodes".sepaGripper.sequence.status.seqActive AND "Unit1.Em7.ControlNodes".sepaGripper."step".transition1[1731] THEN
       "Unit1.Em7.ControlNodes".sepaGripper.sequence.status.nextStep := #JOB_17_STEP_90;
   END_IF;
END_REGION

REGION Network 93: Step[1790] : Job[17] Step End
   RUNG wire#powerrail
      { S7_Templates := "SrcType := DInt" } EQ_Contact(in1 := "Unit1.Em7.ControlNodes".sepaGripper.sequence.status.currentStep, in2 := #JOB_17_STEP_90)
      Contact( "Unit1.Em7.ControlNodes".sepaGripper.sequence.status.seqActive )
      wire#w1
      Coil( "Unit1.Em7.ControlNodes".sepaGripper."step".action1[1790] )
   END_RUNG
   RUNG wire#w1
      Coil( "Unit1.Em7.ControlNodes".sepaGripper."step".transition1[1790] )
   END_RUNG
   RUNG wire#w1
      Contact( "Unit1.Em7.ControlNodes".sepaGripper."step".transition1[1790] )
      Move(in := #STEP_IDLE, out1 => "Unit1.Em7.ControlNodes".sepaGripper.sequence.status.nextStep)
   END_RUNG
   // the same network as SCL:
   "Unit1.Em7.ControlNodes".sepaGripper."step".action1[1790] := ("Unit1.Em7.ControlNodes".sepaGripper.sequence.status.currentStep = #JOB_17_STEP_90) AND "Unit1.Em7.ControlNodes".sepaGripper.sequence.status.seqActive;
   "Unit1.Em7.ControlNodes".sepaGripper."step".transition1[1790] := ("Unit1.Em7.ControlNodes".sepaGripper.sequence.status.currentStep = #JOB_17_STEP_90) AND "Unit1.Em7.ControlNodes".sepaGripper.sequence.status.seqActive;
   IF ("Unit1.Em7.ControlNodes".sepaGripper.sequence.status.currentStep = #JOB_17_STEP_90) AND "Unit1.Em7.ControlNodes".sepaGripper.sequence.status.seqActive AND "Unit1.Em7.ControlNodes".sepaGripper."step".transition1[1790] THEN
       "Unit1.Em7.ControlNodes".sepaGripper.sequence.status.nextStep := #STEP_IDLE;
   END_IF;
END_REGION

REGION Network 94: *************** JOB[18] Return ************************
END_REGION

REGION Network 95: Step[1801] : JOB[18] Condition
   RUNG wire#powerrail
      { S7_Templates := "SrcType := DInt" } EQ_Contact(in1 := "Unit1.Em7.ControlNodes".sepaGripper.sequence.status.currentStep, in2 := #JOB_18_STEP_01)
      Contact( "Unit1.Em7.ControlNodes".sepaGripper.sequence.status.seqActive )
      wire#w1
      Coil( "Unit1.Em7.ControlNodes".sepaGripper."step".action1[1801] )
   END_RUNG
   RUNG wire#w1
      Coil( "Unit1.Em7.ControlNodes".sepaGripper."step".transition1[1801] )
   END_RUNG
   RUNG wire#w1
      Contact( "Unit1.Em7.ControlNodes".sepaGripper."step".transition1[1801] )
      Move(in := #JOB_18_STEP_10, out1 => "Unit1.Em7.ControlNodes".sepaGripper.sequence.status.nextStep)
   END_RUNG
   // the same network as SCL:
   "Unit1.Em7.ControlNodes".sepaGripper."step".action1[1801] := ("Unit1.Em7.ControlNodes".sepaGripper.sequence.status.currentStep = #JOB_18_STEP_01) AND "Unit1.Em7.ControlNodes".sepaGripper.sequence.status.seqActive;
   "Unit1.Em7.ControlNodes".sepaGripper."step".transition1[1801] := ("Unit1.Em7.ControlNodes".sepaGripper.sequence.status.currentStep = #JOB_18_STEP_01) AND "Unit1.Em7.ControlNodes".sepaGripper.sequence.status.seqActive;
   IF ("Unit1.Em7.ControlNodes".sepaGripper.sequence.status.currentStep = #JOB_18_STEP_01) AND "Unit1.Em7.ControlNodes".sepaGripper.sequence.status.seqActive AND "Unit1.Em7.ControlNodes".sepaGripper."step".transition1[1801] THEN
       "Unit1.Em7.ControlNodes".sepaGripper.sequence.status.nextStep := #JOB_18_STEP_10;
   END_IF;
END_REGION

REGION Network 96: Step[1810] : Gripper X-Axis Turn/DisCharge Pos
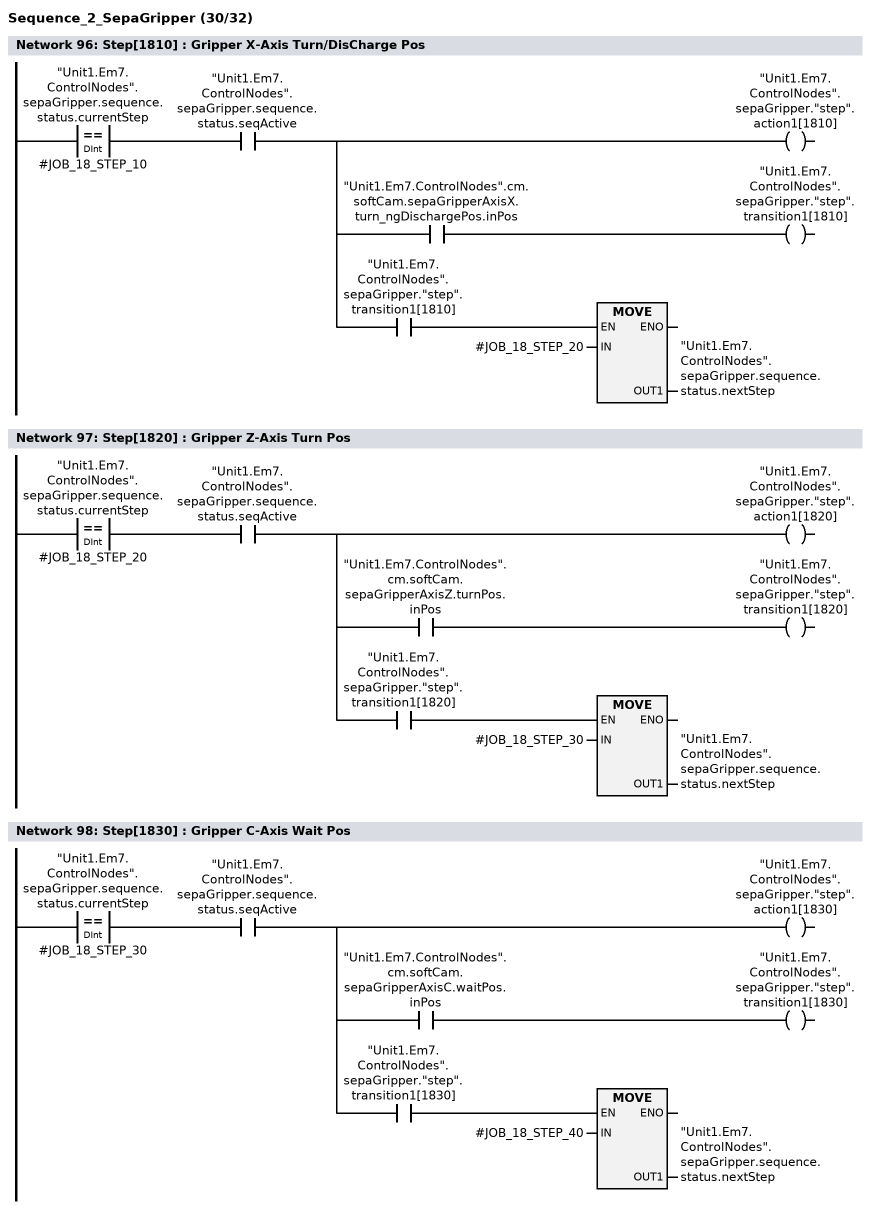
   RUNG wire#powerrail
      { S7_Templates := "SrcType := DInt" } EQ_Contact(in1 := "Unit1.Em7.ControlNodes".sepaGripper.sequence.status.currentStep, in2 := #JOB_18_STEP_10)
      Contact( "Unit1.Em7.ControlNodes".sepaGripper.sequence.status.seqActive )
      wire#w1
      Coil( "Unit1.Em7.ControlNodes".sepaGripper."step".action1[1810] )
   END_RUNG
   RUNG wire#w1
      Contact( "Unit1.Em7.ControlNodes".cm.softCam.sepaGripperAxisX.turn_ngDischargePos.inPos )
      Coil( "Unit1.Em7.ControlNodes".sepaGripper."step".transition1[1810] )
   END_RUNG
   RUNG wire#w1
      Contact( "Unit1.Em7.ControlNodes".sepaGripper."step".transition1[1810] )
      Move(in := #JOB_18_STEP_20, out1 => "Unit1.Em7.ControlNodes".sepaGripper.sequence.status.nextStep)
   END_RUNG
   // the same network as SCL:
   "Unit1.Em7.ControlNodes".sepaGripper."step".action1[1810] := ("Unit1.Em7.ControlNodes".sepaGripper.sequence.status.currentStep = #JOB_18_STEP_10) AND "Unit1.Em7.ControlNodes".sepaGripper.sequence.status.seqActive;
   "Unit1.Em7.ControlNodes".sepaGripper."step".transition1[1810] := ("Unit1.Em7.ControlNodes".sepaGripper.sequence.status.currentStep = #JOB_18_STEP_10) AND "Unit1.Em7.ControlNodes".sepaGripper.sequence.status.seqActive AND "Unit1.Em7.ControlNodes".cm.softCam.sepaGripperAxisX.turn_ngDischargePos.inPos;
   IF ("Unit1.Em7.ControlNodes".sepaGripper.sequence.status.currentStep = #JOB_18_STEP_10) AND "Unit1.Em7.ControlNodes".sepaGripper.sequence.status.seqActive AND "Unit1.Em7.ControlNodes".sepaGripper."step".transition1[1810] THEN
       "Unit1.Em7.ControlNodes".sepaGripper.sequence.status.nextStep := #JOB_18_STEP_20;
   END_IF;
END_REGION

REGION Network 97: Step[1820] : Gripper Z-Axis Turn Pos
   RUNG wire#powerrail
      { S7_Templates := "SrcType := DInt" } EQ_Contact(in1 := "Unit1.Em7.ControlNodes".sepaGripper.sequence.status.currentStep, in2 := #JOB_18_STEP_20)
      Contact( "Unit1.Em7.ControlNodes".sepaGripper.sequence.status.seqActive )
      wire#w1
      Coil( "Unit1.Em7.ControlNodes".sepaGripper."step".action1[1820] )
   END_RUNG
   RUNG wire#w1
      Contact( "Unit1.Em7.ControlNodes".cm.softCam.sepaGripperAxisZ.turnPos.inPos )
      Coil( "Unit1.Em7.ControlNodes".sepaGripper."step".transition1[1820] )
   END_RUNG
   RUNG wire#w1
      Contact( "Unit1.Em7.ControlNodes".sepaGripper."step".transition1[1820] )
      Move(in := #JOB_18_STEP_30, out1 => "Unit1.Em7.ControlNodes".sepaGripper.sequence.status.nextStep)
   END_RUNG
   // the same network as SCL:
   "Unit1.Em7.ControlNodes".sepaGripper."step".action1[1820] := ("Unit1.Em7.ControlNodes".sepaGripper.sequence.status.currentStep = #JOB_18_STEP_20) AND "Unit1.Em7.ControlNodes".sepaGripper.sequence.status.seqActive;
   "Unit1.Em7.ControlNodes".sepaGripper."step".transition1[1820] := ("Unit1.Em7.ControlNodes".sepaGripper.sequence.status.currentStep = #JOB_18_STEP_20) AND "Unit1.Em7.ControlNodes".sepaGripper.sequence.status.seqActive AND "Unit1.Em7.ControlNodes".cm.softCam.sepaGripperAxisZ.turnPos.inPos;
   IF ("Unit1.Em7.ControlNodes".sepaGripper.sequence.status.currentStep = #JOB_18_STEP_20) AND "Unit1.Em7.ControlNodes".sepaGripper.sequence.status.seqActive AND "Unit1.Em7.ControlNodes".sepaGripper."step".transition1[1820] THEN
       "Unit1.Em7.ControlNodes".sepaGripper.sequence.status.nextStep := #JOB_18_STEP_30;
   END_IF;
END_REGION

REGION Network 98: Step[1830] : Gripper C-Axis Wait Pos
   RUNG wire#powerrail
      { S7_Templates := "SrcType := DInt" } EQ_Contact(in1 := "Unit1.Em7.ControlNodes".sepaGripper.sequence.status.currentStep, in2 := #JOB_18_STEP_30)
      Contact( "Unit1.Em7.ControlNodes".sepaGripper.sequence.status.seqActive )
      wire#w1
      Coil( "Unit1.Em7.ControlNodes".sepaGripper."step".action1[1830] )
   END_RUNG
   RUNG wire#w1
      Contact( "Unit1.Em7.ControlNodes".cm.softCam.sepaGripperAxisC.waitPos.inPos )
      Coil( "Unit1.Em7.ControlNodes".sepaGripper."step".transition1[1830] )
   END_RUNG
   RUNG wire#w1
      Contact( "Unit1.Em7.ControlNodes".sepaGripper."step".transition1[1830] )
      Move(in := #JOB_18_STEP_40, out1 => "Unit1.Em7.ControlNodes".sepaGripper.sequence.status.nextStep)
   END_RUNG
   // the same network as SCL:
   "Unit1.Em7.ControlNodes".sepaGripper."step".action1[1830] := ("Unit1.Em7.ControlNodes".sepaGripper.sequence.status.currentStep = #JOB_18_STEP_30) AND "Unit1.Em7.ControlNodes".sepaGripper.sequence.status.seqActive;
   "Unit1.Em7.ControlNodes".sepaGripper."step".transition1[1830] := ("Unit1.Em7.ControlNodes".sepaGripper.sequence.status.currentStep = #JOB_18_STEP_30) AND "Unit1.Em7.ControlNodes".sepaGripper.sequence.status.seqActive AND "Unit1.Em7.ControlNodes".cm.softCam.sepaGripperAxisC.waitPos.inPos;
   IF ("Unit1.Em7.ControlNodes".sepaGripper.sequence.status.currentStep = #JOB_18_STEP_30) AND "Unit1.Em7.ControlNodes".sepaGripper.sequence.status.seqActive AND "Unit1.Em7.ControlNodes".sepaGripper."step".transition1[1830] THEN
       "Unit1.Em7.ControlNodes".sepaGripper.sequence.status.nextStep := #JOB_18_STEP_40;
   END_IF;
END_REGION

REGION Network 99: Step[1840] : Gripper X-Axis Wait Pos
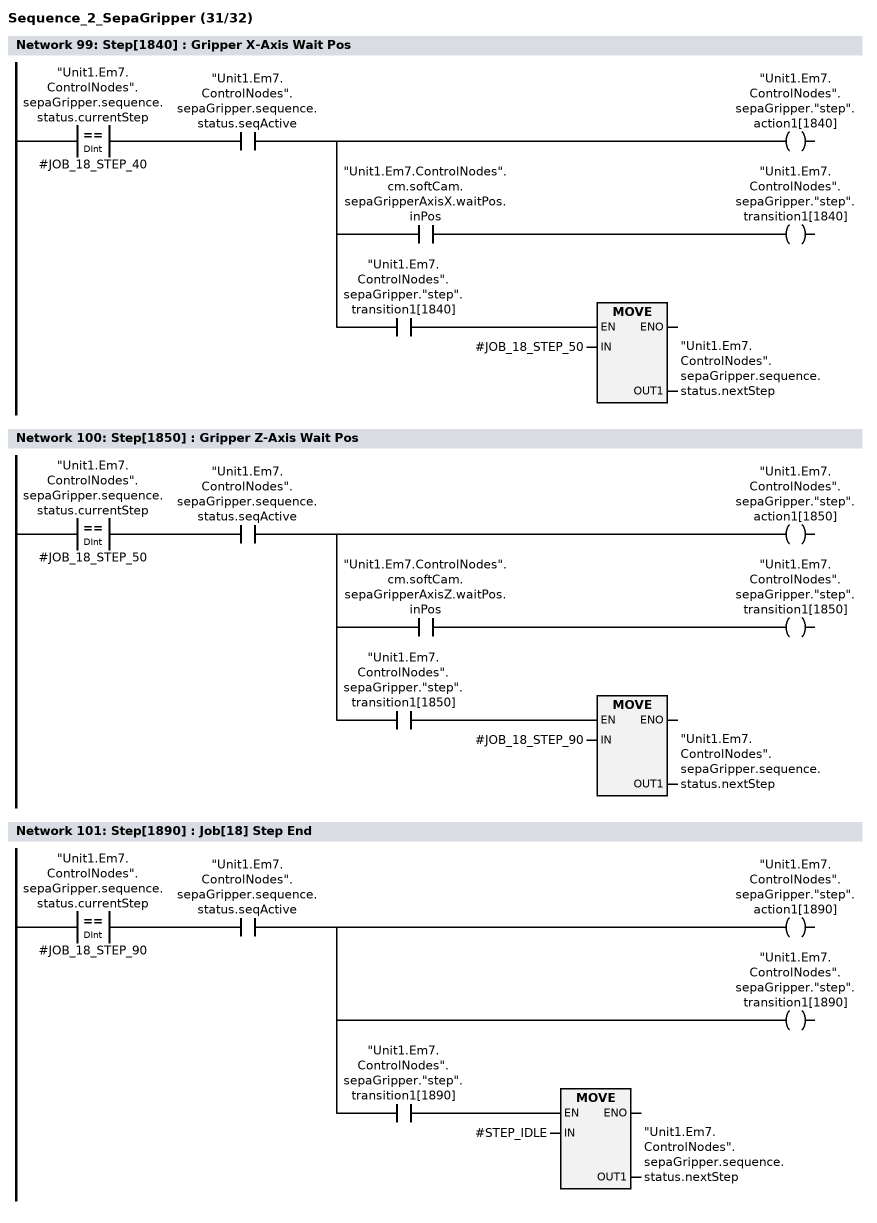
   RUNG wire#powerrail
      { S7_Templates := "SrcType := DInt" } EQ_Contact(in1 := "Unit1.Em7.ControlNodes".sepaGripper.sequence.status.currentStep, in2 := #JOB_18_STEP_40)
      Contact( "Unit1.Em7.ControlNodes".sepaGripper.sequence.status.seqActive )
      wire#w1
      Coil( "Unit1.Em7.ControlNodes".sepaGripper."step".action1[1840] )
   END_RUNG
   RUNG wire#w1
      Contact( "Unit1.Em7.ControlNodes".cm.softCam.sepaGripperAxisX.waitPos.inPos )
      Coil( "Unit1.Em7.ControlNodes".sepaGripper."step".transition1[1840] )
   END_RUNG
   RUNG wire#w1
      Contact( "Unit1.Em7.ControlNodes".sepaGripper."step".transition1[1840] )
      Move(in := #JOB_18_STEP_50, out1 => "Unit1.Em7.ControlNodes".sepaGripper.sequence.status.nextStep)
   END_RUNG
   // the same network as SCL:
   "Unit1.Em7.ControlNodes".sepaGripper."step".action1[1840] := ("Unit1.Em7.ControlNodes".sepaGripper.sequence.status.currentStep = #JOB_18_STEP_40) AND "Unit1.Em7.ControlNodes".sepaGripper.sequence.status.seqActive;
   "Unit1.Em7.ControlNodes".sepaGripper."step".transition1[1840] := ("Unit1.Em7.ControlNodes".sepaGripper.sequence.status.currentStep = #JOB_18_STEP_40) AND "Unit1.Em7.ControlNodes".sepaGripper.sequence.status.seqActive AND "Unit1.Em7.ControlNodes".cm.softCam.sepaGripperAxisX.waitPos.inPos;
   IF ("Unit1.Em7.ControlNodes".sepaGripper.sequence.status.currentStep = #JOB_18_STEP_40) AND "Unit1.Em7.ControlNodes".sepaGripper.sequence.status.seqActive AND "Unit1.Em7.ControlNodes".sepaGripper."step".transition1[1840] THEN
       "Unit1.Em7.ControlNodes".sepaGripper.sequence.status.nextStep := #JOB_18_STEP_50;
   END_IF;
END_REGION

REGION Network 100: Step[1850] : Gripper Z-Axis Wait Pos
   RUNG wire#powerrail
      { S7_Templates := "SrcType := DInt" } EQ_Contact(in1 := "Unit1.Em7.ControlNodes".sepaGripper.sequence.status.currentStep, in2 := #JOB_18_STEP_50)
      Contact( "Unit1.Em7.ControlNodes".sepaGripper.sequence.status.seqActive )
      wire#w1
      Coil( "Unit1.Em7.ControlNodes".sepaGripper."step".action1[1850] )
   END_RUNG
   RUNG wire#w1
      Contact( "Unit1.Em7.ControlNodes".cm.softCam.sepaGripperAxisZ.waitPos.inPos )
      Coil( "Unit1.Em7.ControlNodes".sepaGripper."step".transition1[1850] )
   END_RUNG
   RUNG wire#w1
      Contact( "Unit1.Em7.ControlNodes".sepaGripper."step".transition1[1850] )
      Move(in := #JOB_18_STEP_90, out1 => "Unit1.Em7.ControlNodes".sepaGripper.sequence.status.nextStep)
   END_RUNG
   // the same network as SCL:
   "Unit1.Em7.ControlNodes".sepaGripper."step".action1[1850] := ("Unit1.Em7.ControlNodes".sepaGripper.sequence.status.currentStep = #JOB_18_STEP_50) AND "Unit1.Em7.ControlNodes".sepaGripper.sequence.status.seqActive;
   "Unit1.Em7.ControlNodes".sepaGripper."step".transition1[1850] := ("Unit1.Em7.ControlNodes".sepaGripper.sequence.status.currentStep = #JOB_18_STEP_50) AND "Unit1.Em7.ControlNodes".sepaGripper.sequence.status.seqActive AND "Unit1.Em7.ControlNodes".cm.softCam.sepaGripperAxisZ.waitPos.inPos;
   IF ("Unit1.Em7.ControlNodes".sepaGripper.sequence.status.currentStep = #JOB_18_STEP_50) AND "Unit1.Em7.ControlNodes".sepaGripper.sequence.status.seqActive AND "Unit1.Em7.ControlNodes".sepaGripper."step".transition1[1850] THEN
       "Unit1.Em7.ControlNodes".sepaGripper.sequence.status.nextStep := #JOB_18_STEP_90;
   END_IF;
END_REGION

REGION Network 101: Step[1890] : Job[18] Step End
   RUNG wire#powerrail
      { S7_Templates := "SrcType := DInt" } EQ_Contact(in1 := "Unit1.Em7.ControlNodes".sepaGripper.sequence.status.currentStep, in2 := #JOB_18_STEP_90)
      Contact( "Unit1.Em7.ControlNodes".sepaGripper.sequence.status.seqActive )
      wire#w1
      Coil( "Unit1.Em7.ControlNodes".sepaGripper."step".action1[1890] )
   END_RUNG
   RUNG wire#w1
      Coil( "Unit1.Em7.ControlNodes".sepaGripper."step".transition1[1890] )
   END_RUNG
   RUNG wire#w1
      Contact( "Unit1.Em7.ControlNodes".sepaGripper."step".transition1[1890] )
      Move(in := #STEP_IDLE, out1 => "Unit1.Em7.ControlNodes".sepaGripper.sequence.status.nextStep)
   END_RUNG
   // the same network as SCL:
   "Unit1.Em7.ControlNodes".sepaGripper."step".action1[1890] := ("Unit1.Em7.ControlNodes".sepaGripper.sequence.status.currentStep = #JOB_18_STEP_90) AND "Unit1.Em7.ControlNodes".sepaGripper.sequence.status.seqActive;
   "Unit1.Em7.ControlNodes".sepaGripper."step".transition1[1890] := ("Unit1.Em7.ControlNodes".sepaGripper.sequence.status.currentStep = #JOB_18_STEP_90) AND "Unit1.Em7.ControlNodes".sepaGripper.sequence.status.seqActive;
   IF ("Unit1.Em7.ControlNodes".sepaGripper.sequence.status.currentStep = #JOB_18_STEP_90) AND "Unit1.Em7.ControlNodes".sepaGripper.sequence.status.seqActive AND "Unit1.Em7.ControlNodes".sepaGripper."step".transition1[1890] THEN
       "Unit1.Em7.ControlNodes".sepaGripper.sequence.status.nextStep := #STEP_IDLE;
   END_IF;
END_REGION

REGION Network 102: *************** IMMEDIATE STOP **************************
END_REGION

REGION Network 103: Immediate Stop
END_REGION

REGION Network 104: *************** Status updates **************************
END_REGION

REGION Network 105: Sequence Status
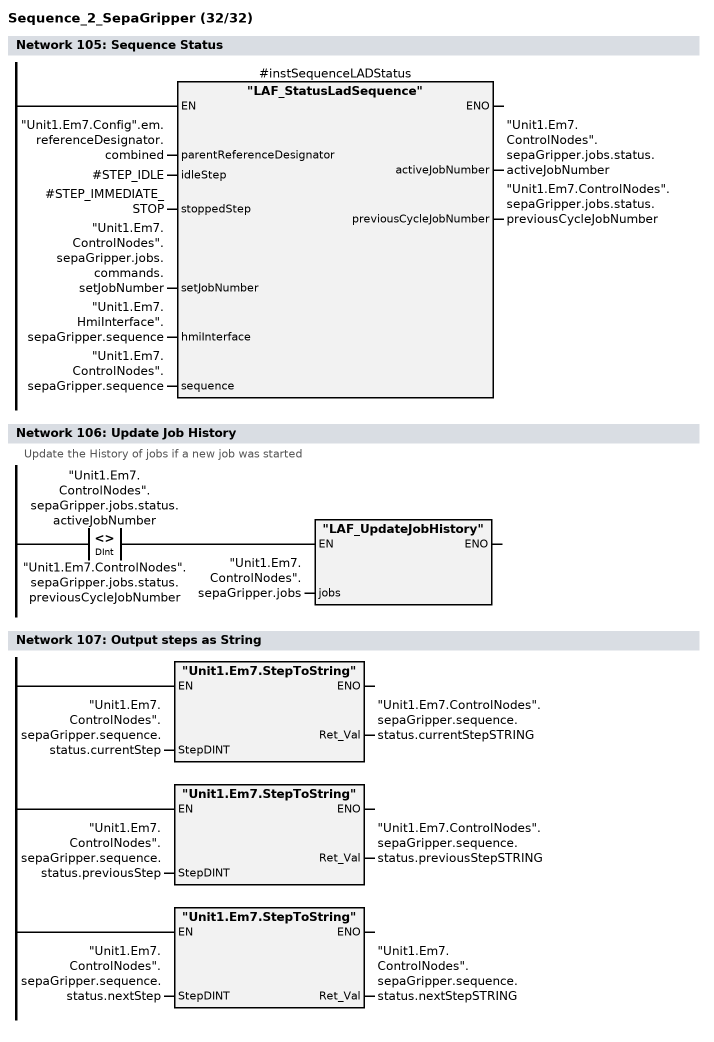
   RUNG wire#powerrail
      #instSequenceLADStatus(parentReferenceDesignator := "Unit1.Em7.Config".em.referenceDesignator.combined, idleStep := #STEP_IDLE, stoppedStep := #STEP_IMMEDIATE_STOP, setJobNumber := "Unit1.Em7.ControlNodes".sepaGripper.jobs.commands.setJobNumber, hmiInterface := "Unit1.Em7.HmiInterface".sepaGripper.sequence, sequence := "Unit1.Em7.ControlNodes".sepaGripper.sequence, activeJobNumber => "Unit1.Em7.ControlNodes".sepaGripper.jobs.status.activeJobNumber, previousCycleJobNumber => "Unit1.Em7.ControlNodes".sepaGripper.jobs.status.previousCycleJobNumber)
   END_RUNG
   // the same network as SCL:
   #instSequenceLADStatus(parentReferenceDesignator := "Unit1.Em7.Config".em.referenceDesignator.combined,   // "LAF_StatusLadSequence"
                          idleStep := #STEP_IDLE,
                          stoppedStep := #STEP_IMMEDIATE_STOP,
                          setJobNumber := "Unit1.Em7.ControlNodes".sepaGripper.jobs.commands.setJobNumber,
                          hmiInterface := "Unit1.Em7.HmiInterface".sepaGripper.sequence,
                          sequence := "Unit1.Em7.ControlNodes".sepaGripper.sequence,
                          activeJobNumber => "Unit1.Em7.ControlNodes".sepaGripper.jobs.status.activeJobNumber,
                          previousCycleJobNumber => "Unit1.Em7.ControlNodes".sepaGripper.jobs.status.previousCycleJobNumber);
END_REGION

REGION Network 106: Update Job History
   // Update the History of jobs if a new job was started
   RUNG wire#powerrail
      { S7_Templates := "SrcType := DInt" } NE_Contact(in1 := "Unit1.Em7.ControlNodes".sepaGripper.jobs.status.activeJobNumber, in2 := "Unit1.Em7.ControlNodes".sepaGripper.jobs.status.previousCycleJobNumber)
      "LAF_UpdateJobHistory"(jobs := "Unit1.Em7.ControlNodes".sepaGripper.jobs)
   END_RUNG
   // the same network as SCL:
   IF "Unit1.Em7.ControlNodes".sepaGripper.jobs.status.activeJobNumber <> "Unit1.Em7.ControlNodes".sepaGripper.jobs.status.previousCycleJobNumber THEN
       "LAF_UpdateJobHistory"(jobs := "Unit1.Em7.ControlNodes".sepaGripper.jobs);
   END_IF;
END_REGION

REGION Network 107: Output steps as String
   RUNG wire#powerrail
      "Unit1.Em7.StepToString"(StepDINT := "Unit1.Em7.ControlNodes".sepaGripper.sequence.status.currentStep, Ret_Val => "Unit1.Em7.ControlNodes".sepaGripper.sequence.status.currentStepSTRING)
   END_RUNG
   RUNG wire#powerrail
      "Unit1.Em7.StepToString"(StepDINT := "Unit1.Em7.ControlNodes".sepaGripper.sequence.status.previousStep, Ret_Val => "Unit1.Em7.ControlNodes".sepaGripper.sequence.status.previousStepSTRING)
   END_RUNG
   RUNG wire#powerrail
      "Unit1.Em7.StepToString"(StepDINT := "Unit1.Em7.ControlNodes".sepaGripper.sequence.status.nextStep, Ret_Val => "Unit1.Em7.ControlNodes".sepaGripper.sequence.status.nextStepSTRING)
   END_RUNG
   // the same network as SCL:
   "Unit1.Em7.ControlNodes".sepaGripper.sequence.status.currentStepSTRING := "Unit1.Em7.StepToString"(StepDINT := "Unit1.Em7.ControlNodes".sepaGripper.sequence.status.currentStep);
   "Unit1.Em7.ControlNodes".sepaGripper.sequence.status.previousStepSTRING := "Unit1.Em7.StepToString"(StepDINT := "Unit1.Em7.ControlNodes".sepaGripper.sequence.status.previousStep);
   "Unit1.Em7.ControlNodes".sepaGripper.sequence.status.nextStepSTRING := "Unit1.Em7.StepToString"(StepDINT := "Unit1.Em7.ControlNodes".sepaGripper.sequence.status.nextStep);
END_REGION
END_FUNCTION_BLOCK
